(* IEC 61131-3 sources: B-R/Processes/EDT, 38 files *)

(* ---- EDTP1S1_1_ACTION.st ---- *)
ACTION P1S1_1_ACT:
	//步与步之间切换的设定时间,至少设置为5s(可更改，调整阀门到位、液位延时后),用于检查步骤错误信号
	FOR i := 0 TO EDTP1S1_1_STEP_NUM DO
		IF EDTP1S1_1_ST[i] < T#5s THEN
			EDTP1S1_1_ST[i] := T#5s;
		END_IF;
		EDTP1S1_1_STEP[i].set_time := EDTP1S1_1_ST[i];
	END_FOR;

	//流程步骤
	ProcessHandleFC(EDTP1S1_1,EDTP1S1_1_STEP[0],EDTP1S1_1_STEP_NUM);

	//object 手自动切换
	IF (EDTP1S1_1.status.mode <> 0) AND (NOT EDTP1S1_1.auto_mode_edge) THEN
		EDTP1S1_1.auto_mode_edge := TRUE;
		EDTP1S1_1.manual_mode_edge := FALSE;
		EDTR01.control.auto_operate := TRUE;
		EDTFQV0502.control.auto_operate := TRUE;
		EDTXV0505.control.auto_operate := TRUE;
	END_IF;

	IF (EDTP1S1_1.status.mode = 0) AND (NOT EDTP1S1_1.manual_mode_edge) THEN
		EDTP1S1_1.manual_mode_edge := TRUE;
		EDTP1S1_1.auto_mode_edge := FALSE;
		EDTR01.control.manual_operate := TRUE;
		EDTFQV0502.control.manual_operate := TRUE;
		EDTXV0505.control.manual_operate := TRUE;
	END_IF;

	//错误信号停机
	EDTP1S1_1.input.error_signal := (EDTR01.status.motor_status >= 2) OR (EDTFQV0502.status.valve_status >= 2) OR
	(EDTXV0505.status.valve_status >= 2);

	//步骤执行动作
	IF EDTP1S1_1.status.run_state = 1 THEN
		CASE EDTP1S1_1.status.run_step OF
			0:
				//初始化检查
				IF NOT EDTP1S1_1_STEP[0].done THEN
					EDTR01.control.auto_operate := TRUE;
					EDTFQV0502.control.auto_operate := TRUE;
					EDTXV0505.control.auto_operate := TRUE;
					EDTP1S1_1_STEP[0].done := TRUE;
				END_IF;
			1:
				//关闭底阀
				EDTXV0505.input.auto_open_signal := FALSE;
				IF EDTXV0505.input.close_feedback_state THEN
					EDTP1S1_1_STEP[1].done := TRUE;
				END_IF;
			2:
				//加定量纯水
				LiquidTransfer_3(sp_time := DINT_TO_TIME(EDTP1S1_1_PARA_T1 * 1000),
				sp_accumulation := EDTP1S1_1_PARA_AC1,
				done := EDTP1S1_1_STEP[2].done,
				flowmeter := EDTFQIT1904);
				EDTFQV0502.input.auto_open_signal := LiquidTransfer_3.run;
			3:
				//开启搅拌
				EDTR01.input.auto_run_signal := TRUE;
				IF EDTR01.input.run_feedback THEN
					EDTP1S1_1_STEP[3].done := TRUE;
				END_IF;
			4:
				//人工投料，完成后点击确认
			5:
				//溶解计时
				TON_41.PT := DINT_TO_TIME(EDTP1S1_1_PARA_T2 * 60 * 1000);
				TON_41.IN := TRUE;
				IF TON_41.Q THEN
					TON_41.IN := FALSE;
					EDTP1S1_1_STEP[5].done := TRUE;
				END_IF;
				TON_41();
			6:
				//观察溶解结束后点击确认
		END_CASE;
	END_IF;

	//人工确认步骤可用
	IF (EDTP1S1_1.status.run_state) AND (NOT EDTP1S1_1_STEP[EDTP1S1_1.status.run_step].done AND ((EDTP1S1_1.status.run_step = 4) OR (EDTP1S1_1.status.run_step = 6))) THEN
		EDTP1S1_1.status.confirm_enable := TRUE;
	ELSE
		EDTP1S1_1.status.confirm_enable := FALSE;
	END_IF;
END_ACTION

(* ---- EDTP1S1_ACTION.st ---- *)
ACTION P1S1_ACT:
	//步与步之间切换的设定时间,至少设置为5s(可更改，调整阀门到位、液位延时后),用于检查步骤错误信号
	FOR i := 0 TO EDTP1S1_STEP_NUM DO
		IF EDTP1S1_ST[i] < T#5s THEN
			EDTP1S1_ST[i] := T#5s;
		END_IF;
		EDTP1S1_STEP[i].set_time := EDTP1S1_ST[i];
	END_FOR;

	//流程步骤
	ProcessHandleFC(EDTP1S1,EDTP1S1_STEP[0],EDTP1S1_STEP_NUM);

	//object 手自动切换
	IF (EDTP1S1.status.mode <> 0) AND (NOT EDTP1S1.auto_mode_edge) THEN
		EDTP1S1.auto_mode_edge := TRUE;
		EDTP1S1.manual_mode_edge := FALSE;
		EDTR02.control.auto_operate := TRUE;
		EDTFQV0101.control.auto_operate := TRUE;
		EDTXV0102.control.auto_operate := TRUE;
	END_IF;

	IF (EDTP1S1.status.mode = 0) AND (NOT EDTP1S1.manual_mode_edge) THEN
		EDTP1S1.manual_mode_edge := TRUE;
		EDTP1S1.auto_mode_edge := FALSE;
		EDTR02.control.manual_operate := TRUE;
		EDTFQV0101.control.manual_operate := TRUE;
		EDTXV0102.control.manual_operate := TRUE;
	END_IF;

	//错误信号停机
	EDTP1S1.input.error_signal := (EDTR02.status.motor_status >= 2) OR (EDTFQV0101.status.valve_status >= 2) OR
	(EDTXV0102.status.valve_status >= 2);

	//步骤执行动作
	IF EDTP1S1.status.run_state = 1 THEN
		CASE EDTP1S1.status.run_step OF
			0:
				//初始化检查
				IF NOT EDTP1S1_STEP[0].done THEN
					EDTR02.control.auto_operate := TRUE;
					EDTFQV0101.control.auto_operate := TRUE;
					EDTXV0102.control.auto_operate := TRUE;
					EDTP1S1_STEP[0].done := TRUE;
				END_IF;
			1:
				//关底阀
				EDTXV0102.input.auto_open_signal := FALSE;
				IF EDTXV0102.input.close_feedback_state THEN
					EDTP1S1_STEP[1].done := TRUE;
				END_IF;
			2:
				//加定量纯水
				LiquidTransfer_0(sp_time := DINT_TO_TIME(EDTP1S1_PARA_T1 * 1000),
				sp_accumulation := EDTP1S1_PARA_AC1,
				done := EDTP1S1_STEP[2].done,
				flowmeter := EDTFQIT1904);
				EDTFQV0101.input.auto_open_signal := LiquidTransfer_0.run;
			3:
				//开启搅拌
				EDTR02.input.auto_run_signal := TRUE;
				IF EDTR02.input.run_feedback THEN
					EDTP1S1_STEP[3].done := TRUE;
				END_IF;
			4:
				//人工投料，完成后点击确认
			5:
				//溶解计时
				TON_49.PT := DINT_TO_TIME(EDTP1S1_PARA_T2 * 60 * 1000);
				TON_49.IN := TRUE;
				IF TON_49.Q THEN
					TON_49.IN := FALSE;
					EDTP1S1_STEP[5].done := TRUE;
				END_IF;
				TON_49();
			6:
				//观察溶解结束
			7:
				//开底阀，关搅拌
				EDTXV0102.input.auto_open_signal := TRUE;
				IF EDTXV0102.input.open_feedback_state THEN
					EDTR02.input.auto_run_signal := FALSE;
					IF NOT EDTR02.input.run_feedback THEN
						EDTP1S1_STEP[7].done := TRUE;
					END_IF;
				END_IF;
			8:
				//观察釜内放料完成，点击确认
			9:
				EDTXV0102.input.auto_open_signal := FALSE;
				IF EDTXV0102.input.close_feedback_state THEN
					EDTP1S1_STEP[9].done := TRUE;
				END_IF;
			10:
				//手动通氮气清理过滤器
		END_CASE;
	END_IF;

	//人工确认步骤可用
	IF (EDTP1S1.status.run_state) AND (NOT EDTP1S1_STEP[EDTP1S1.status.run_step].done AND ((EDTP1S1.status.run_step = 4) OR (EDTP1S1.status.run_step = 6)
		OR (EDTP1S1.status.run_step = 8) OR (EDTP1S1.status.run_step = 10))) THEN
		EDTP1S1.status.confirm_enable := TRUE;
	ELSE
		EDTP1S1.status.confirm_enable := FALSE;
	END_IF;
END_ACTION

(* ---- EDTP1S2A_ACTION.st ---- *)
ACTION P1S2A_ACT:
	//设定时间
	FOR i := 0 TO EDTP1S2_STEP_NUM DO
		IF EDTP1S2A_ST[i] < T#5s THEN
			EDTP1S2A_ST[i] := T#5s;
		END_IF;
		EDTP1S2A_STEP[i].set_time := EDTP1S2A_ST[i];
	END_FOR;

	//流程步骤
	ProcessHandleFC(EDTP1S2A,EDTP1S2A_STEP[0],EDTP1S2_STEP_NUM);

	//object 手自动切换
	IF (EDTP1S2A.status.mode <> 0) AND (NOT EDTP1S2A.auto_mode_edge) THEN

		EDTP1S2A.auto_mode_edge := TRUE;
		EDTP1S2A.manual_mode_edge := FALSE;

		EDTP01.control.auto_operate := TRUE;
		EDTXV0205.control.auto_operate := TRUE;
		STFLV0701.control.auto_operate := TRUE;
		STFLV0702.control.auto_operate := TRUE;
		EDTLV0201.control.auto_operate := TRUE;
		STFP07.control.auto_operate := TRUE;
		EDTR07A.control.auto_operate := TRUE;
		EDTTV0201A.control.auto_operate := TRUE;
		EDTTV0201B.control.auto_operate := TRUE;
		EDTXV0201.control.auto_operate := TRUE;
		EDTXV0204.control.auto_operate := TRUE;
		EDTXV0505.control.auto_operate := TRUE;
		EDTFQV0203A.control.auto_operate := TRUE;
		EDTP26.control.auto_operate := TRUE;
	END_IF;

	IF (EDTP1S2A.status.mode = 0) AND (NOT EDTP1S2A.manual_mode_edge) THEN

		EDTP1S2A.manual_mode_edge := TRUE;
		EDTP1S2A.auto_mode_edge := FALSE;

		EDTP01.control.manual_operate := TRUE;
		EDTXV0205.control.manual_operate := TRUE;
		STFLV0701.control.manual_operate := TRUE;
		STFLV0702.control.manual_operate := TRUE;
		EDTLV0201.control.manual_operate := TRUE;
		STFP07.control.manual_operate := TRUE;
		EDTR07A.control.manual_operate := TRUE;
		EDTTV0201A.control.manual_operate := TRUE;
		EDTTV0201B.control.manual_operate := TRUE;
		EDTXV0201.control.manual_operate := TRUE;
		EDTXV0204.control.manual_operate := TRUE;
		EDTXV0505.control.manual_operate := TRUE;
		EDTFQV0203A.control.manual_operate := TRUE;
		EDTP26.control.manual_operate := TRUE;
	END_IF;

	//错误信号停机
	EDTP1S2A.input.error_signal := (EDTP01.status.motor_status >= 2) OR (EDTXV0205.status.valve_status >= 2) OR
	(STFLV0701.status.valve_status >= 2) OR (STFLV0702.status.valve_status >= 2) OR (EDTLV0201.status.valve_status >= 2) OR
	(STFP07.status.motor_status >= 2) OR (EDTR07A.status.motor_status >= 2) OR
	(EDTTV0201A.status.valve_status >= 2) OR (EDTTV0201B.status.valve_status >= 2) OR (EDTXV0201.status.valve_status >= 2) OR
	(EDTP26.status.motor_status >= 2) OR (EDTFQV0203A.status.valve_status >= 2) OR (EDTXV0505.status.valve_status >= 2) OR
	(EDTXV0204.status.valve_status >= 2);

	IF EDTP1S2A.status.run_state = 1 THEN
		CASE EDTP1S2A.status.run_step OF
			0:
				//初始化
				IF NOT EDTP1S2A_STEP[0].done THEN
					EDTP01.control.auto_operate := TRUE;
					EDTXV0205.control.auto_operate := TRUE;
					STFLV0701.control.auto_operate := TRUE;
					STFLV0702.control.auto_operate := TRUE;
					EDTLV0201.control.auto_operate := TRUE;
					STFP07.control.auto_operate := TRUE;
					EDTR07A.control.auto_operate := TRUE;
					EDTTV0201A.control.auto_operate := TRUE;
					EDTTV0201B.control.auto_operate := TRUE;
					EDTXV0201.control.auto_operate := TRUE;
					EDTXV0204.control.auto_operate := TRUE;
					EDTXV0505.control.auto_operate := TRUE;
					EDTFQV0203A.control.auto_operate := TRUE;
					EDTP26.control.auto_operate := TRUE;
					EDTP1S2A_STEP[0].done := TRUE;
				END_IF;
			1:
				//人工确认投料
			2:
				//滴加
				CASE p1_step2_2a OF
					0:
						IF NOT EDTP1S2A_STEP[2].done THEN
							p1_step2_2a := 1;
						END_IF;
					1:
						EDTXV0201.input.auto_open_signal := TRUE;
						EDTR07A.input.auto_run_signal := TRUE;
						IF EDTXV0201.input.open_feedback_state AND EDTR07A.input.run_feedback THEN
							p1_step2_2a := 2;
						END_IF;
					2:
						IF EDTTIT0201.status.value <= EDTP1S2_PARA_Temp1 THEN
							p1_step2_2a := 3;
						END_IF;
					3:
						TON_2.PT := DINT_TO_TIME(EDTP1S2_PARA_T5 * 60 * 1000);
						TON_2.IN := TRUE;
						IF EDTTIT0201.status.value <= EDTP1S2_PARA_Temp2 THEN
							EDTTV0201A.input.auto_open_signal := TRUE;
							EDTTV0201B.input.auto_open_signal := TRUE;
						END_IF;
						IF EDTTIT0201.status.value >= EDTP1S2_PARA_Temp3 THEN
							EDTTV0201A.input.auto_open_signal := FALSE;
							EDTTV0201B.input.auto_open_signal := FALSE;
						END_IF;
						IF TON_2.Q THEN
							TON_2.IN := FALSE;
							EDTXV0201.input.auto_open_signal := FALSE;
							EDTTV0201A.input.auto_open_signal := TRUE;
							EDTTV0201B.input.auto_open_signal := TRUE;
							p1_step2_2a := 4;
						END_IF;
					4:
						TON_2.PT := DINT_TO_TIME(EDTP1S2_PARA_T6 * 60 * 1000);
						TON_2.IN := TRUE;
						IF TON_2.Q THEN
							TON_2.IN := FALSE;
							EDTTV0201A.input.auto_open_signal := FALSE;
							EDTTV0201B.input.auto_open_signal := FALSE;
							p1_step2_2a := 5;
						END_IF;
					5:
						IF EDTTV0201A.input.close_feedback_state AND EDTTV0201B.input.close_feedback_state THEN
							EDTP1S2A_STEP[2].done := TRUE;
							p1_step2_2a := 0;
						END_IF;
				END_CASE;
				TON_2();
			3:
				//取样确认
			4:
				TON_9.PT := DINT_TO_TIME(EDTP1S2_PARA_T7 * 60 * 1000);
				EDTR07A.input.auto_run_signal := FALSE;
				IF NOT EDTR07A.input.run_feedback THEN
					TON_9.IN := TRUE;
				END_IF;
				IF TON_9.Q THEN
					TON_9.IN := FALSE;
					EDTP1S2A_STEP[4].done := TRUE;
				END_IF;
				TON_9();
		END_CASE;
	END_IF;

	//R07A进ABC溶液
	IF r07a_add THEN
		CASE p1_step2_4a OF
			0:
				EDTXV0204.input.auto_open_signal := FALSE;
				EDTXV0201.input.auto_open_signal := TRUE;
				IF EDTXV0204.input.close_feedback_state AND EDTXV0201.input.open_feedback_state THEN
					p1_step2_4a := 1;
				END_IF;
			1:
				EDTXV0505.input.auto_open_signal := TRUE;
				EDTFQV0203A.input.auto_open_signal := TRUE;
				IF EDTXV0505.input.open_feedback_state AND EDTFQV0203A.input.open_feedback_state THEN
					p1_step2_4a := 2;
				END_IF;
			2:
			//等待液体充满泵后，再启动P26防止抽空。
				TON_54.PT := DINT_TO_TIME(EDTP1S2A_PARA_T4 * 1000);
				TON_54.IN := TRUE;
				IF TON_54.Q THEN
					TON_54.IN := FALSE;
					p1_step2_4a := 3;
				END_IF;
			3:
				LiquidTransfer_4(sp_time := DINT_TO_TIME(EDTP1S2A_PARA_T8 * 1000),
				sp_accumulation := EDTP1S2A_PARA_AC2,
				done := p1_step2_4a_3_done,
				flowmeter := EDTFQIT0203);
				EDTP26.input.auto_run_signal := LiquidTransfer_4.run;
				IF p1_step2_4a_3_done AND (NOT EDTP26.input.run_feedback) AND (NOT EDTP26.input.auto_run_signal) THEN
					p1_step2_4a := 4;
					p1_step2_4a_3_done := FALSE;
				END_IF;
			4:
				IF EDTFQIT0203.flowrate <= flowrate_threshold THEN
					EDTXV0505.input.auto_open_signal := FALSE;
					EDTFQV0203A.input.auto_open_signal := FALSE;
				END_IF;
				IF EDTXV0505.input.close_feedback_state AND EDTFQV0203A.input.close_feedback_state THEN
					r07a_add := FALSE;
					p1_step2_4a := 0;
				END_IF;
		END_CASE;
		TON_54();
	END_IF;

	//V02A（SSS溶液）进料
	IF v02a_add THEN
		CASE p1_step2_1a OF
			0:
				p1_step2_1a := 1;
			1:
				EDTXV0205.input.auto_open_signal := TRUE;
				IF EDTXV0205.input.open_feedback_state THEN
					p1_step2_1a := 2;
				END_IF;
			2:
				LiquidAddSimple_0(level_value := EDTLIT0203.status.value,
				sp_value := EDTP1S2A_PARA_L2,
				sp_time := DINT_TO_TIME(EDTP1S2A_PARA_T1 * 60 * 1000),
				done := p1_step2_1a_2_done);
				EDTP01.input.auto_run_signal := LiquidAddSimple_0.run;
				IF p1_step2_1a_2_done AND (NOT EDTP01.input.run_feedback) AND (NOT EDTP01.input.auto_run_signal) THEN
					p1_step2_1a := 3;
					p1_step2_1a_2_done := FALSE;
				END_IF;
			3:
				TON_1.PT := DINT_TO_TIME(EDTP1S2A_PARA_T2 * 1000);
				TON_1.IN := TRUE;
				IF TON_1.Q THEN
					TON_1.IN := FALSE;
					p1_step2_1a := 4;
				END_IF;
			4:
				EDTXV0205.input.auto_open_signal := FALSE;
				IF EDTXV0205.input.close_feedback_state THEN
					v02a_add := FALSE;
					p1_step2_1a := 0;
				END_IF;
		END_CASE;
		TON_1();
	END_IF;

	//V03A（MCE）进料
	IF v03a_add THEN
		CASE p1_step2_3a OF
			0:
				p1_step2_3a := 1;
			1:
				STFLV0702.input.auto_open_signal := FALSE;
				STFLV0701.input.auto_open_signal := FALSE;
				EDTLV0201.input.auto_open_signal := TRUE;
				IF EDTLV0201.input.open_feedback_state AND STFLV0701.input.close_feedback_state
					AND STFLV0702.input.close_feedback_state THEN
					p1_step2_3a := 2;
				END_IF;
			2:
				LiquidAdd_3(level_value := EDTLIT0201.status.value,
				sp_value := EDTP1S2A_PARA_L1,
				sp_accumulation := EDTP1S2A_PARA_AC1,
				sp_time := DINT_TO_TIME(EDTP1S2A_PARA_T3 * 1000),
				flowmeter := STFFQIT0702,
				done := p1_step2_3a_2_done);
				STFP07.input.auto_run_signal := LiquidAdd_3.run;
				IF p1_step2_3a_2_done AND (NOT STFP07.input.run_feedback) AND (NOT STFP07.input.auto_run_signal) THEN
					p1_step2_3a := 3;
				END_IF;
			3:
				IF STFFQIT0702.flowrate <= flowrate_threshold THEN
					EDTLV0201.input.auto_open_signal := FALSE;
				END_IF;
				IF EDTLV0201.input.close_feedback_state THEN
					p1_step2_3a_2_done := FALSE;
					p1_step2_3a := 0;
					v03a_add := FALSE;
				END_IF;
		END_CASE;
	END_IF;
		//人工确认步骤可用
		IF (EDTP1S2A.status.run_state) AND (NOT EDTP1S2A_STEP[EDTP1S2A.status.run_step].done AND ((EDTP1S2A.status.run_step = 1) OR (EDTP1S2A.status.run_step = 3))) THEN
			EDTP1S2A.status.confirm_enable := TRUE;
		ELSE
			EDTP1S2A.status.confirm_enable := FALSE;
		END_IF;
		END_ACTION

(* ---- EDTP1S2B_ACTION.st ---- *)
ACTION P1S2B_ACT:
	//设定时间
	FOR i := 0 TO EDTP1S2_STEP_NUM DO
		IF EDTP1S2B_ST[i] < T#5s THEN
			EDTP1S2B_ST[i] := T#5s;
		END_IF;
		EDTP1S2B_STEP[i].set_time := EDTP1S2B_ST[i];
	END_FOR;

	//流程步骤
	ProcessHandleFC(EDTP1S2B,EDTP1S2B_STEP[0],EDTP1S2_STEP_NUM);

	//object 手自动切换
	IF (EDTP1S2B.status.mode <> 0) AND (NOT EDTP1S2B.auto_mode_edge) THEN

		EDTP1S2B.auto_mode_edge := TRUE;
		EDTP1S2B.manual_mode_edge := FALSE;

		EDTP01.control.auto_operate := TRUE;
		EDTXV0206.control.auto_operate := TRUE;
		STFLV0701.control.auto_operate := TRUE;
		STFLV0702.control.auto_operate := TRUE;
		EDTLV0202.control.auto_operate := TRUE;
		STFP07.control.auto_operate := TRUE;
		EDTR07B.control.auto_operate := TRUE;
		EDTTV0202A.control.auto_operate := TRUE;
		EDTTV0202B.control.auto_operate := TRUE;
		EDTXV0202.control.auto_operate := TRUE;
		EDTXV0203.control.auto_operate := TRUE;
		EDTXV0505.control.auto_operate := TRUE;
		EDTFQV0203B.control.auto_operate := TRUE;
		EDTP26.control.auto_operate := TRUE;
	END_IF;

	IF (EDTP1S2B.status.mode = 0) AND (NOT EDTP1S2B.manual_mode_edge) THEN

		EDTP1S2B.manual_mode_edge := TRUE;
		EDTP1S2B.auto_mode_edge := FALSE;

		EDTP01.control.manual_operate := TRUE;
		EDTXV0206.control.manual_operate := TRUE;
		STFLV0701.control.manual_operate := TRUE;
		STFLV0702.control.manual_operate := TRUE;
		EDTLV0202.control.manual_operate := TRUE;
		STFP07.control.manual_operate := TRUE;
		EDTR07B.control.manual_operate := TRUE;
		EDTTV0202A.control.manual_operate := TRUE;
		EDTTV0202B.control.manual_operate := TRUE;
		EDTXV0202.control.manual_operate := TRUE;
		EDTXV0203.control.manual_operate := TRUE;
		EDTXV0505.control.manual_operate := TRUE;
		EDTFQV0203B.control.manual_operate := TRUE;
		EDTP26.control.manual_operate := TRUE;
	END_IF;

	//错误信号停机
	EDTP1S2B.input.error_signal := (EDTP01.status.motor_status >= 2) OR (EDTXV0206.status.valve_status >= 2) OR
	(STFLV0701.status.valve_status >= 2) OR (STFLV0702.status.valve_status >= 2) OR (EDTLV0202.status.valve_status >= 2) OR
	(STFP07.status.motor_status >= 2) OR (EDTR07B.status.motor_status >= 2) OR
	(EDTTV0202A.status.valve_status >= 2) OR (EDTTV0202B.status.valve_status >= 2) OR (EDTXV0202.status.valve_status >= 2) OR
	(EDTP26.status.motor_status >= 2) OR (EDTFQV0203B.status.valve_status >= 2) OR (EDTXV0505.status.valve_status >= 2) OR
	(EDTXV0203.status.valve_status >= 2);

	IF EDTP1S2B.status.run_state = 1 THEN
		CASE EDTP1S2B.status.run_step OF
			0:
				//初始化
				IF NOT EDTP1S2B_STEP[0].done THEN
					EDTP01.control.auto_operate := TRUE;
					EDTXV0206.control.auto_operate := TRUE;
					STFLV0701.control.auto_operate := TRUE;
					STFLV0702.control.auto_operate := TRUE;
					EDTLV0202.control.auto_operate := TRUE;
					STFP07.control.auto_operate := TRUE;
					EDTR07B.control.auto_operate := TRUE;
					EDTTV0202A.control.auto_operate := TRUE;
					EDTTV0202B.control.auto_operate := TRUE;
					EDTXV0202.control.auto_operate := TRUE;
					EDTXV0203.control.auto_operate := TRUE;
					EDTXV0505.control.auto_operate := TRUE;
					EDTFQV0203B.control.auto_operate := TRUE;
					EDTP26.control.auto_operate := TRUE;
					EDTP1S2B_STEP[0].done := TRUE;
				END_IF;
			1:
				//人工确认投料
			2:
				//滴加
				CASE p1_step2_2b OF
					0:
						IF NOT EDTP1S2B_STEP[2].done THEN
							p1_step2_2b := 1;
						END_IF;
					1:
						EDTXV0202.input.auto_open_signal := TRUE;
						EDTR07B.input.auto_run_signal := TRUE;
						IF EDTXV0202.input.open_feedback_state AND EDTR07B.input.run_feedback THEN
							p1_step2_2b := 2;
						END_IF;
					2:
						IF EDTTIT0202.status.value <= EDTP1S2_PARA_Temp1 THEN
							p1_step2_2b := 3;
						END_IF;
					3:
						TON_5.PT := DINT_TO_TIME(EDTP1S2_PARA_T5 * 60 * 1000);
						TON_5.IN := TRUE;
						IF EDTTIT0202.status.value <= EDTP1S2_PARA_Temp2 THEN
							EDTTV0202A.input.auto_open_signal := TRUE;
							EDTTV0202B.input.auto_open_signal := TRUE;
						END_IF;
						IF EDTTIT0202.status.value >= EDTP1S2_PARA_Temp3 THEN
							EDTTV0202A.input.auto_open_signal := FALSE;
							EDTTV0202B.input.auto_open_signal := FALSE;
						END_IF;
						IF TON_5.Q THEN
							TON_5.IN := FALSE;
							EDTXV0202.input.auto_open_signal := FALSE;
							EDTTV0202A.input.auto_open_signal := TRUE;
							EDTTV0202B.input.auto_open_signal := TRUE;
							p1_step2_2b := 4;
						END_IF;
					4:
						TON_5.PT := DINT_TO_TIME(EDTP1S2_PARA_T6 * 60 * 1000);
						TON_5.IN := TRUE;
						IF TON_5.Q THEN
							TON_5.IN := FALSE;
							EDTTV0202A.input.auto_open_signal := FALSE;
							EDTTV0202B.input.auto_open_signal := FALSE;
							p1_step2_2b := 5;
						END_IF;
					5:
						IF EDTTV0202A.input.close_feedback_state AND EDTTV0202B.input.close_feedback_state THEN
							EDTP1S2B_STEP[2].done := TRUE;
							p1_step2_2b := 0;
						END_IF;
				END_CASE;
				TON_5();
			3:
				//取样确认
			4:
				TON_18.PT := DINT_TO_TIME(EDTP1S2_PARA_T7 * 60 * 1000);
				EDTR07B.input.auto_run_signal := FALSE;
				IF NOT EDTR07B.input.run_feedback THEN
					TON_18.IN := TRUE;
				END_IF;
				IF TON_18.Q THEN
					TON_18.IN := FALSE;
					EDTP1S2B_STEP[4].done := TRUE;
				END_IF;
				TON_18();
		END_CASE;
	END_IF;

	//R07A进ABC溶液
	IF r07b_add THEN
		CASE p1_step2_4b OF
			0:
				EDTXV0203.input.auto_open_signal := FALSE;
				EDTXV0202.input.auto_open_signal := TRUE;
				IF EDTXV0203.input.close_feedback_state AND EDTXV0202.input.open_feedback_state THEN
					p1_step2_4b := 1;
				END_IF;
			1:
				EDTXV0505.input.auto_open_signal := TRUE;
				EDTFQV0203B.input.auto_open_signal := TRUE;
				IF EDTXV0505.input.open_feedback_state AND EDTFQV0203B.input.open_feedback_state THEN
					p1_step2_4b := 2;
				END_IF;
			2:
				//等待液体充满泵后，再启动P26防止抽空。
				TON_55.PT := DINT_TO_TIME(EDTP1S2B_PARA_T4 * 1000);
				TON_55.IN := TRUE;
				IF TON_55.Q THEN
					TON_55.IN := FALSE;
					p1_step2_4b := 3;
				END_IF;
			3:
				LiquidTransfer_5(sp_time := DINT_TO_TIME(EDTP1S2B_PARA_T8 * 1000),
				sp_accumulation := EDTP1S2B_PARA_AC2,
				done := p1_step2_4b_3_done,
				flowmeter := EDTFQIT0203);
				EDTP26.input.auto_run_signal := LiquidTransfer_5.run;
				IF p1_step2_4b_3_done AND (NOT EDTP26.input.run_feedback) AND (NOT EDTP26.input.auto_run_signal) THEN
					p1_step2_4b := 4;
					p1_step2_4b_3_done := FALSE;
				END_IF;
			4:
				IF EDTFQIT0203.flowrate <= flowrate_threshold THEN
					EDTXV0505.input.auto_open_signal := FALSE;
					EDTFQV0203B.input.auto_open_signal := FALSE;
				END_IF;
				IF EDTXV0505.input.close_feedback_state AND EDTFQV0203B.input.close_feedback_state THEN
					r07b_add := FALSE;
					p1_step2_4b := 0;
				END_IF;
		END_CASE;
		TON_55();
	END_IF;

	//V02B（SSS溶液）进料
	IF v02b_add THEN
		CASE p1_step2_1b OF
			0:
				p1_step2_1b := 1;
			1:
				EDTXV0206.input.auto_open_signal := TRUE;
				IF EDTXV0206.input.open_feedback_state THEN
					p1_step2_1b := 2;
				END_IF;
			2:
				LiquidAddSimple_1(level_value := EDTLIT0204.status.value,
				sp_value := EDTP1S2B_PARA_L2,
				sp_time := DINT_TO_TIME(EDTP1S2B_PARA_T1 * 60 * 1000),
				done := p1_step2_1b_2_done);
				EDTP01.input.auto_run_signal := LiquidAddSimple_1.run;
				IF p1_step2_1b_2_done AND (NOT EDTP01.input.run_feedback) AND (NOT EDTP01.input.auto_run_signal) THEN
					p1_step2_1b := 3;
					p1_step2_1b_2_done := FALSE;
				END_IF;
			3:
				TON_4.PT := DINT_TO_TIME(EDTP1S2B_PARA_T2 * 1000);
				TON_4.IN := TRUE;
				IF TON_4.Q THEN
					TON_4.IN := FALSE;
					p1_step2_1b := 4;
				END_IF;
			4:
				EDTXV0206.input.auto_open_signal := FALSE;
				IF EDTXV0206.input.close_feedback_state THEN
					v02b_add := FALSE;
					p1_step2_1b := 0;
				END_IF;
		END_CASE;
		TON_4();
	END_IF;

	//V03B（MCE）进料
	IF v03b_add THEN
		CASE p1_step2_3b OF
			0:
				p1_step2_3b := 1;
			1:
				STFLV0702.input.auto_open_signal := FALSE;
				STFLV0701.input.auto_open_signal := FALSE;
				EDTLV0202.input.auto_open_signal := TRUE;
				IF EDTLV0202.input.open_feedback_state AND STFLV0701.input.close_feedback_state
					AND STFLV0702.input.close_feedback_state THEN
					p1_step2_3b := 2;
				END_IF;
			2:
				LiquidAdd_5(level_value := EDTLIT0202.status.value,
				sp_value := EDTP1S2B_PARA_L1,
				sp_accumulation := EDTP1S2B_PARA_AC1,
				sp_time := DINT_TO_TIME(EDTP1S2B_PARA_T3 * 1000),
				flowmeter := STFFQIT0702,
				done := p1_step2_3b_2_done);
				STFP07.input.auto_run_signal := LiquidAdd_5.run;
				IF p1_step2_3b_2_done AND (NOT STFP07.input.run_feedback) AND (NOT STFP07.input.auto_run_signal) THEN
					p1_step2_3b := 3;
				END_IF;
			3:
				IF STFFQIT0702.flowrate <= flowrate_threshold THEN
					EDTLV0202.input.auto_open_signal := FALSE;
				END_IF;
				IF EDTLV0202.input.close_feedback_state THEN
					p1_step2_3b_2_done := FALSE;
					p1_step2_3b := 0;
					v03b_add := FALSE;
				END_IF;
		END_CASE;
	END_IF;

	//人工确认步骤可用
	IF (EDTP1S2B.status.run_state) AND (NOT EDTP1S2B_STEP[EDTP1S2B.status.run_step].done AND ((EDTP1S2B.status.run_step = 1) OR (EDTP1S2B.status.run_step = 3))) THEN
		EDTP1S2B.status.confirm_enable := TRUE;
	ELSE
		EDTP1S2B.status.confirm_enable := FALSE;
	END_IF;
		END_ACTION

(* ---- EDTP1S3_ACTION.st ---- *)
ACTION P1S3_ACT:
	//设定时间
	FOR i := 0 TO EDTP1S3_STEP_NUM DO
		IF EDTP1S3_ST[i] < T#5s THEN
			EDTP1S3_ST[i] := T#5s;
		END_IF;
		EDTP1S3_STEP[i].set_time := EDTP1S3_ST[i];
	END_FOR;

	//流程步骤
	ProcessHandleFC(EDTP1S3,EDTP1S3_STEP[0],EDTP1S3_STEP_NUM);

	//object 手自动切换
	IF (EDTP1S3.status.mode <> 0) AND (NOT EDTP1S3.auto_mode_edge) THEN
		EDTP1S3.auto_mode_edge := TRUE;
		EDTP1S3.manual_mode_edge := FALSE;

		EDTXV0304.control.auto_operate := TRUE;
		EDTXV0410.control.auto_operate := TRUE;
		EDTXV0302.control.auto_operate := TRUE;
		EDTTV0301G.control.auto_operate := TRUE;
		EDTR13.control.auto_operate := TRUE;
		EDTP03.control.auto_operate := TRUE;
		EDTTV0301C.control.auto_operate := TRUE;
		EDTTV0301D.control.auto_operate := TRUE;
		EDTTV0301E.control.auto_operate := TRUE;
		EDTTV0301F.control.auto_operate := TRUE;
		EDTTV0301A.control.auto_operate := TRUE;
		EDTTV0301B.control.auto_operate := TRUE;
		EDTPV0301.control.auto_operate := TRUE;
	END_IF;

	IF (EDTP1S3.status.mode = 0) AND (NOT EDTP1S3.manual_mode_edge) THEN
		EDTP1S3.manual_mode_edge := TRUE;
		EDTP1S3.auto_mode_edge := FALSE;

		EDTXV0304.control.manual_operate := TRUE;
		EDTXV0410.control.manual_operate := TRUE;
		EDTXV0302.control.manual_operate := TRUE;
		EDTTV0301G.control.manual_operate := TRUE;
		EDTR13.control.manual_operate := TRUE;
		EDTP03.control.manual_operate := TRUE;
		EDTTV0301C.control.manual_operate := TRUE;
		EDTTV0301D.control.manual_operate := TRUE;
		EDTTV0301E.control.manual_operate := TRUE;
		EDTTV0301F.control.manual_operate := TRUE;
		EDTTV0301A.control.manual_operate := TRUE;
		EDTTV0301B.control.manual_operate := TRUE;
		EDTPV0301.control.manual_operate := TRUE;
	END_IF;

	//错误信号停机
	EDTP1S3.input.error_signal :=
	(EDTXV0304.status.valve_status >= 2) OR (EDTXV0410.status.valve_status >= 2) OR (EDTXV0302.status.valve_status >= 2) OR
	(EDTTV0301G.status.valve_status >= 2) OR (EDTR13.status.motor_status >= 2) OR
	(EDTP03.status.motor_status >= 2) OR (EDTTV0301C.status.valve_status >= 2) OR
	(EDTTV0301D.status.valve_status >= 2) OR (EDTTV0301E.status.valve_status >= 2) OR
	(EDTTV0301F.status.valve_status >= 2) OR (EDTTV0301A.status.valve_status >= 2) OR
	(EDTTV0301B.status.valve_status >= 2) OR (EDTPV0301.status.valve_status >= 2);

	IF EDTP1S3.status.run_state = 1 THEN
		CASE EDTP1S3.status.run_step OF
			0:
				//初始化
				IF NOT EDTP1S3_STEP[0].done THEN
					EDTXV0302.control.auto_operate := TRUE;
					EDTXV0304.control.auto_operate := TRUE;
					EDTXV0410.control.auto_operate := TRUE;
					EDTTV0301G.control.auto_operate := TRUE;
					EDTR13.control.auto_operate := TRUE;
					EDTP03.control.auto_operate := TRUE;
					EDTTV0301C.control.auto_operate := TRUE;
					EDTTV0301D.control.auto_operate := TRUE;
					EDTTV0301E.control.auto_operate := TRUE;
					EDTTV0301F.control.auto_operate := TRUE;
					EDTTV0301A.control.auto_operate := TRUE;
					EDTTV0301B.control.auto_operate := TRUE;
					EDTPV0301.control.auto_operate := TRUE;
					EDTP1S3_STEP[0].done := TRUE;
				END_IF;
			1:
				//确认R13釜空闲,手动开阀进料
			2:
				EDTXV0302.input.auto_open_signal := TRUE;
				IF EDTXV0302.input.open_feedback_state THEN
					EDTXV0304.input.auto_open_signal := TRUE;
				END_IF;
				IF EDTXV0304.input.open_feedback_state THEN
					EDTTV0301G.input.auto_open_signal := TRUE;
				END_IF;
				IF EDTTV0301G.input.open_feedback_state THEN
					EDTXV0410.input.auto_open_signal := TRUE;
				END_IF;
				IF EDTXV0302.input.open_feedback_state AND EDTXV0304.input.open_feedback_state AND EDTTV0301G.input.open_feedback_state
					AND EDTXV0410.input.open_feedback_state THEN
					EDTR13.input.auto_run_signal := TRUE;
					EDTP03.input.auto_run_signal := TRUE;
					IF EDTR13.input.run_feedback AND EDTP03.input.run_feedback THEN
						EDTP1S3_STEP[2].done := TRUE;
					END_IF;
				END_IF;
			3:
				CASE p1_step3_3 OF
					0:
						IF NOT EDTP1S3_STEP[3].done THEN
							p1_step3_3 := 1;
						END_IF;
					1:
						HeatPot_0(ST1 := DINT_TO_TIME(EDTP1S3_PARA_T1 * 1000),
						ST2 := DINT_TO_TIME(EDTP1S3_PARA_T2 * 1000),
						V3 := EDTTV0301C,
						V4 := EDTTV0301D,
						V5 := EDTTV0301E,
						V6 := EDTTV0301F,
						done := p1_step3_3_1_done);
						IF p1_step3_3_1_done THEN
							p1_step3_3 := 2;
						END_IF;
					2:
						IF EDTTIT0301.status.value >= EDTP1S3_PARA_Temp1 THEN
							EDTTV0301C.input.auto_open_signal := FALSE;
							IF EDTTIT0301.status.value >= EDTP1S3_PARA_Temp2 THEN
								p1_step3_3 := 3;
							END_IF;
						END_IF;
					3:
						TON_40.PT := DINT_TO_TIME(EDTP1S3_PARA_T3 * 60 * 1000);
						TON_40.IN := TRUE;
						IF TON_40.Q THEN
							TON_40.IN := FALSE;
							EDTTV0301D.input.auto_open_signal := FALSE;
							EDTTV0301E.input.auto_open_signal := FALSE;
							p1_step3_3 := 4;
						END_IF;
					4:
						TON_40.PT := DINT_TO_TIME(EDTP1S3_PARA_T4 * 60 * 1000);
						TON_40.IN := TRUE;
						IF TON_40.Q THEN
							TON_40.IN := FALSE;
							EDTTV0301F.input.auto_open_signal := TRUE;
							p1_step3_3 := 5;
						END_IF;
					5:
						TON_40.PT := DINT_TO_TIME(EDTP1S3_PARA_T5 * 1000);
						TON_40.IN := TRUE;
						IF TON_40.Q THEN
							TON_40.IN := FALSE;
							EDTTV0301F.input.auto_open_signal := FALSE;
							p1_step3_3 := 6;
						END_IF;
					6:
						IF EDTTV0301C.input.close_feedback_state AND EDTTV0301D.input.close_feedback_state AND EDTTV0301E.input.close_feedback_state AND EDTTV0301F.input.close_feedback_state THEN
							p1_step3_3 := 0;
							p1_step3_3_1_done := FALSE;
							EDTP1S3_STEP[3].done := TRUE;
						END_IF;
				END_CASE;
				TON_40();
			4:
				CASE p1_step3_4 OF
					0:
						IF NOT EDTP1S3_STEP[4].done THEN
							p1_step3_4 := 1;
						END_IF;
					1:
						EDTTV0301A.input.auto_open_signal := TRUE;
						IF EDTTV0301A.input.open_feedback_state THEN
							EDTTV0301B.input.auto_open_signal := TRUE;
							IF EDTTV0301B.input.open_feedback_state THEN
								p1_step3_4 := 2;
							END_IF;
						END_IF;
					2:
						IF EDTTIT0301.status.value <= EDTP1S3_PARA_Temp4 THEN
							EDTPV0301.input.auto_open_signal := TRUE;
							p1_step3_4 := 3;
						END_IF;
					3:
						IF EDTPIT0301.status.value >= EDTP1S3_PARA_P1 THEN
							EDTTV0301G.input.auto_open_signal := FALSE;
							IF EDTTV0301G.input.close_feedback_state THEN
								EDTP03.input.auto_run_signal := FALSE;
								p1_step3_4 := 4;
							END_IF;
						END_IF;
					4:
						IF NOT EDTP03.input.run_feedback THEN
							EDTXV0410.input.auto_open_signal := FALSE;
							EDTXV0304.input.auto_open_signal := FALSE;
							EDTTV0301A.input.auto_open_signal := FALSE;
							EDTTV0301B.input.auto_open_signal := FALSE;
							p1_step3_4 := 5;
						END_IF;
					5:
						IF EDTPIT0301.status.value >= EDTP1S3_PARA_P2 THEN
							EDTXV0302.input.auto_open_signal := FALSE;
							EDTPV0301.input.auto_open_signal := FALSE;
							EDTR13.input.auto_run_signal := FALSE;
							EDTP1S3_STEP[4].done := TRUE;
							p1_step3_4 := 0;
						END_IF;
				END_CASE;
		END_CASE;
	END_IF;

	//人工确认步骤可用
	IF (EDTP1S3.status.run_state) AND (NOT EDTP1S3_STEP[EDTP1S3.status.run_step].done AND ((EDTP1S3.status.run_step = 1))) THEN
		EDTP1S3.status.confirm_enable := TRUE;
	ELSE
		EDTP1S3.status.confirm_enable := FALSE;
	END_IF;
END_ACTION

(* ---- EDTP1S4_ACTION.st ---- *)
ACTION P1S4_ACT:
	//设定时间
	FOR i := 0 TO EDTP1S4_STEP_NUM DO
		IF EDTP1S4_ST[i] < T#5s THEN
			EDTP1S4_ST[i] := T#5s;
		END_IF;
		EDTP1S4_STEP[i].set_time := EDTP1S4_ST[i];
	END_FOR;

	//流程步骤
	ProcessHandleFC(EDTP1S4,EDTP1S4_STEP[0],EDTP1S4_STEP_NUM);

	//object 手自动切换
	IF (EDTP1S4.status.mode <> 0) AND (NOT EDTP1S4.auto_mode_edge) THEN
		EDTP1S4.auto_mode_edge := TRUE;
		EDTP1S4.manual_mode_edge := FALSE;

		EDTLV0401.control.auto_operate := TRUE;
		STFP14.control.auto_operate := TRUE;
		STFLV1401.control.auto_operate := TRUE;
		STFLV1402.control.auto_operate := TRUE;
		EDTXV0404.control.auto_operate := TRUE;
		EDTXV0405.control.auto_operate := TRUE;
	END_IF;

	IF (EDTP1S4.status.mode = 0) AND (NOT EDTP1S4.manual_mode_edge) THEN
		EDTP1S4.manual_mode_edge := TRUE;
		EDTP1S4.auto_mode_edge := FALSE;

		EDTLV0401.control.manual_operate := TRUE;
		STFP14.control.manual_operate := TRUE;
		STFLV1401.control.manual_operate := TRUE;
		STFLV1402.control.manual_operate := TRUE;
		EDTXV0404.control.manual_operate := TRUE;
		EDTXV0405.control.manual_operate := TRUE;
	END_IF;

	//错误信号停机
	EDTP1S4.input.error_signal := (EDTXV0405.status.valve_status >= 2) OR (EDTXV0404.status.valve_status >= 2) OR (EDTLV0401.status.valve_status >= 2) OR
	(STFLV1401.status.valve_status >= 2) OR (STFLV1402.status.valve_status >= 2) OR (STFP14.status.motor_status >= 2);

	IF EDTP1S4.status.run_state = 1 THEN
		CASE EDTP1S4.status.run_step OF
			0:
				//初始化
				IF NOT EDTP1S4_STEP[0].done THEN
					EDTLV0401.control.auto_operate := TRUE;
					STFP14.control.auto_operate := TRUE;
					STFLV1401.control.auto_operate := TRUE;
					STFLV1402.control.auto_operate := TRUE;
					EDTXV0404.control.auto_operate := TRUE;
					EDTXV0405.control.auto_operate := TRUE;
					EDTP1S4_STEP[0].done := TRUE;
				END_IF;
		END_CASE;
	END_IF;

	//人工确认步骤可用
//	IF (EDTP1S4.status.run_step = 1) OR (EDTP1S4.status.run_step = 5) THEN
//		EDTP1S4.status.confirm_enable := TRUE;
//	ELSE
//		EDTP1S4.status.confirm_enable := FALSE;
//	END_IF;

	//v07放料
	IF v07_release_start THEN
		CASE v07_release_step OF
			0:
				EDTXV0404.control.auto_operate := TRUE;
				EDTXV0405.control.auto_operate := TRUE;

				EDTXV0405.input.auto_open_signal := TRUE;
				IF EDTXV0405.input.open_feedback_state THEN
					EDTXV0404.input.auto_open_signal := TRUE;
					IF EDTXV0404.input.open_feedback_state THEN
						v07_release_step := 1;
					END_IF;
				END_IF;
			1:
				TON_6.PT := DINT_TO_TIME(EDTP1S4_PARA_T1 * 60 * 1000);
				TON_6.IN := TRUE;
				IF TON_6.Q AND (EDTLIT0401.status.value <= 0.0) THEN
					TON_6.IN := FALSE;
					v07_release_step := 2;
				END_IF;
			2:
				EDTXV0404.input.auto_open_signal := FALSE;
				EDTXV0405.input.auto_open_signal := FALSE;
				IF EDTXV0404.input.close_feedback_state AND EDTXV0405.input.close_feedback_state THEN
					v07_release_step := 3;
				END_IF;
			3:
				v07_release_step := 0;
				v07_release_start := FALSE;
		END_CASE;
		TON_6();
	END_IF;

	//v07进料
	IF v07_add_start THEN
		CASE v07_add_step OF
			0:
				EDTLV0401.control.auto_operate := TRUE;
				STFP14.control.auto_operate := TRUE;
				STFLV1401.control.auto_operate := TRUE;
				STFLV1402.control.auto_operate := TRUE;
				EDTXV0404.control.auto_operate := TRUE;
				EDTXV0405.control.auto_operate := TRUE;

				EDTLV0401.input.auto_open_signal := TRUE;
				EDTXV0405.input.auto_open_signal := TRUE;
				STFLV1401.input.auto_open_signal := TRUE;
				STFLV1402.input.auto_open_signal := FALSE;
				IF EDTLV0401.input.open_feedback_state AND EDTXV0405.input.open_feedback_state AND
					STFLV1401.input.open_feedback_state AND STFLV1402.input.close_feedback_state THEN
					v07_add_step := 1;
				END_IF;
			1:
				LiquidAdd_4(level_value := EDTLIT0401.status.value,
				sp_value := EDTP1S4_PARA_L1,
				sp_accumulation := EDTP1S4_PARA_AC1,
				sp_time := DINT_TO_TIME(EDTP1S4_PARA_T2 * 1000),
				flowmeter := STFFQIT1402,
				done := v07_add_done);
				STFP14.input.auto_run_signal := LiquidAdd_4.run;
				IF v07_add_done AND (NOT STFP14.input.run_feedback) AND (NOT STFP14.input.auto_run_signal) THEN
					v07_add_step := 2;
				END_IF;
			2:
				IF STFFQIT1402.flowrate <= flowrate_threshold THEN
					EDTLV0401.input.auto_open_signal := FALSE;
					EDTXV0405.input.auto_open_signal := FALSE;
					v07_add_step := 3;
				END_IF;
			3:
				v07_add_step := 0;
				v07_add_done := FALSE;
				v07_add_start := FALSE;
		END_CASE;
	END_IF;
END_ACTION

(* ---- EDTP1S5_ACTION.st ---- *)
ACTION P1S5_ACT:
	//设定时间
	FOR i := 0 TO EDTP1S5_STEP_NUM DO
		IF EDTP1S5_ST[i] < T#5s THEN
			EDTP1S5_ST[i] := T#5s;
		END_IF;
		EDTP1S5_STEP[i].set_time := EDTP1S5_ST[i];
	END_FOR;

	//流程步骤
	ProcessHandleFC(EDTP1S5,EDTP1S5_STEP[0],EDTP1S5_STEP_NUM);

	//object 手自动切换
	IF (EDTP1S5.status.mode <> 0) AND (NOT EDTP1S5.auto_mode_edge) THEN
		EDTP1S5.auto_mode_edge := TRUE;
		EDTP1S5.manual_mode_edge := FALSE;

		EDTXV0406.control.auto_operate := TRUE;
		EDTXV0407.control.auto_operate := TRUE;
		EDTXV0410.control.auto_operate := TRUE;
		EDTTV0403G.control.auto_operate := TRUE;
		EDTR19.control.auto_operate := TRUE;
		EDTP03.control.auto_operate := TRUE;
		EDTTV0403A.control.auto_operate := TRUE;
		EDTTV0403B.control.auto_operate := TRUE;
		EDTTV0403C.control.auto_operate := TRUE;
		EDTTV0403D.control.auto_operate := TRUE;
		EDTTV0403E.control.auto_operate := TRUE;
		EDTTV0403F.control.auto_operate := TRUE;
		EDTXV0411.control.auto_operate := TRUE;
		EDTPV0401.control.auto_operate := TRUE;
	END_IF;

	IF (EDTP1S5.status.mode = 0) AND (NOT EDTP1S5.manual_mode_edge) THEN
		EDTP1S5.manual_mode_edge := TRUE;
		EDTP1S5.auto_mode_edge := FALSE;

		EDTXV0406.control.manual_operate := TRUE;
		EDTXV0407.control.manual_operate := TRUE;
		EDTXV0410.control.manual_operate := TRUE;
		EDTTV0403G.control.manual_operate := TRUE;
		EDTR19.control.manual_operate := TRUE;
		EDTP03.control.manual_operate := TRUE;
		EDTTV0403A.control.manual_operate := TRUE;
		EDTTV0403B.control.manual_operate := TRUE;
		EDTTV0403C.control.manual_operate := TRUE;
		EDTTV0403D.control.manual_operate := TRUE;
		EDTTV0403E.control.manual_operate := TRUE;
		EDTTV0403F.control.manual_operate := TRUE;
		EDTXV0411.control.manual_operate := TRUE;
		EDTPV0401.control.manual_operate := TRUE;
	END_IF;

	//错误信号停机
	EDTP1S5.input.error_signal := (EDTXV0406.status.valve_status >= 2) OR (EDTXV0407.status.valve_status >= 2) OR
	(EDTXV0410.status.valve_status >= 2) OR (EDTTV0403G.status.valve_status >= 2) OR
	(EDTR19.status.motor_status >= 2) OR (EDTP03.status.motor_status >= 2) OR (EDTTV0403A.status.valve_status >= 2) OR
	(EDTTV0403B.status.valve_status >= 2) OR (EDTTV0403C.status.valve_status >= 2) OR (EDTTV0403D.status.valve_status >= 2) OR
	(EDTTV0403E.status.valve_status >= 2) OR (EDTTV0403F.status.valve_status >= 2) OR (EDTXV0411.status.valve_status >= 2) OR
	(EDTPV0401.status.valve_status >= 2);

	IF EDTP1S5.status.run_state = 1 THEN
		//步骤执行动作
		CASE EDTP1S5.status.run_step OF
			0:
				//初始化
				IF NOT EDTP1S5_STEP[0].done THEN
					EDTXV0406.control.auto_operate := TRUE;
					EDTXV0407.control.auto_operate := TRUE;
					EDTXV0410.control.auto_operate := TRUE;
					EDTTV0403G.control.auto_operate := TRUE;
					EDTR19.control.auto_operate := TRUE;
					EDTP03.control.auto_operate := TRUE;
					EDTTV0403A.control.auto_operate := TRUE;
					EDTTV0403B.control.auto_operate := TRUE;
					EDTTV0403C.control.auto_operate := TRUE;
					EDTTV0403D.control.auto_operate := TRUE;
					EDTTV0403E.control.auto_operate := TRUE;
					EDTTV0403F.control.auto_operate := TRUE;
					EDTXV0411.control.auto_operate := TRUE;
					EDTPV0401.control.auto_operate := TRUE;
					EDTP1S5_STEP[0].done := TRUE;
				END_IF;
			1:
				//确认V07空闲
			2:
				EDTXV0405.input.auto_open_signal := FALSE;
				IF EDTXV0405.input.close_feedback_state THEN
					EDTXV0406.input.auto_open_signal := TRUE;
				END_IF;
				IF EDTXV0406.input.open_feedback_state THEN
					EDTXV0407.input.auto_open_signal := TRUE;
				END_IF;
				IF EDTXV0407.input.open_feedback_state THEN
					EDTXV0410.input.auto_open_signal := TRUE;
				END_IF;
				IF EDTXV0410.input.open_feedback_state THEN
					EDTTV0403G.input.auto_open_signal := TRUE;
				END_IF;
				IF EDTTV0403G.input.open_feedback_state THEN
					EDTXV0411.input.auto_open_signal := TRUE;
				END_IF;
				IF EDTXV0406.input.open_feedback_state AND EDTXV0407.input.open_feedback_state AND EDTXV0405.input.close_feedback_state
					AND EDTXV0410.input.open_feedback_state AND EDTTV0403G.input.open_feedback_state AND EDTXV0411.input.open_feedback_state THEN
					EDTR19.input.auto_run_signal := TRUE;
					EDTP03.input.auto_run_signal := TRUE;
					IF EDTR19.input.run_feedback AND EDTP03.input.run_feedback THEN
						EDTP1S5_STEP[2].done := TRUE;
					END_IF;
				END_IF;
			3:
				CASE p1_step5_3 OF
					0:
						IF NOT EDTP1S5_STEP[3].done THEN
							p1_step5_3 := 1;
						END_IF;
					1:
						HeatPot_13(ST1 := DINT_TO_TIME(EDTP1S5_PARA_T1 * 1000),
						ST2 := DINT_TO_TIME(EDTP1S5_PARA_T2 * 1000),
						V3 := EDTTV0403C,
						V4 := EDTTV0403D,
						V5 := EDTTV0403E,
						V6 := EDTTV0403F,
						done := p1_step5_3_1_done);
						IF p1_step5_3_1_done THEN
							p1_step5_3_1_done := FALSE;
							p1_step5_3 := 2;
						END_IF;
					2:
						IF EDTTIT0403.status.value >= EDTP1S5_PARA_Temp1 THEN
							EDTTV0403C.input.auto_open_signal := FALSE;
							IF EDTTIT0403.status.value >= EDTP1S5_PARA_Temp2 THEN
								p1_step5_3 := 3;
							END_IF;
						END_IF;
					3:
						TON_45.PT := DINT_TO_TIME(EDTP1S5_PARA_T3 * 60 * 1000);
						TON_45.IN := TRUE;
						IF TON_45.Q THEN
							TON_45.IN := FALSE;
							EDTTV0403D.input.auto_open_signal := FALSE;
							EDTTV0403E.input.auto_open_signal := FALSE;
							p1_step5_3 := 4;
						END_IF;
					4:
						TON_45.PT := DINT_TO_TIME(EDTP1S5_PARA_T4 * 60 * 1000);
						TON_45.IN := TRUE;
						IF TON_45.Q THEN
							TON_45.IN := FALSE;
							EDTTV0403F.input.auto_open_signal := TRUE;
							p1_step5_3 := 5;
						END_IF;
					5:
						TON_45.PT := DINT_TO_TIME(EDTP1S5_PARA_T5 * 1000);
						TON_45.IN := TRUE;
						IF TON_45.Q THEN
							TON_45.IN := FALSE;
							EDTTV0403F.input.auto_open_signal := FALSE;
							p1_step5_3 := 6;
						END_IF;
					6:
						IF EDTTV0403C.input.close_feedback_state AND EDTTV0403D.input.close_feedback_state AND EDTTV0403E.input.close_feedback_state AND EDTTV0403F.input.close_feedback_state THEN
							EDTP1S5_STEP[3].done := TRUE;
							p1_step5_3 := 0;
						END_IF;
				END_CASE;
				TON_45();
			4:
				CASE p1_step5_4 OF
					0:
						IF NOT EDTP1S5_STEP[4].done THEN
							p1_step5_4 := 1;
						END_IF;
					1:
						EDTTV0403A.input.auto_open_signal := TRUE;
						IF	EDTTV0403A.input.open_feedback_state THEN
							EDTTV0403B.input.auto_open_signal := TRUE;
							IF EDTTV0403B.input.open_feedback_state THEN
								p1_step5_4 := 2;
							END_IF;
						END_IF;
					2:
						IF EDTTIT0403.status.value <= EDTP1S5_PARA_Temp4 THEN
							EDTPV0401.input.auto_open_signal := TRUE;
							p1_step5_4 := 3;
						END_IF;
					3:
						IF EDTPIT0401.status.value >= EDTP1S5_PARA_P1 THEN
							EDTTV0403G.input.auto_open_signal := FALSE;
							EDTP03.input.auto_run_signal := FALSE;
							EDTXV0406.input.auto_open_signal := FALSE;
							EDTXV0407.input.auto_open_signal := FALSE;
							EDTXV0410.input.auto_open_signal := FALSE;
							EDTTV0403A.input.auto_open_signal := FALSE;
							EDTTV0403B.input.auto_open_signal := FALSE;
							p1_step5_4 := 4;
						END_IF;
					4:
						IF EDTPIT0401.status.value >= EDTP1S5_PARA_P2 THEN
							EDTPV0401.input.auto_open_signal := FALSE;
							EDTXV0411.input.auto_open_signal := FALSE;
							EDTR19.input.auto_run_signal := FALSE;
							p1_step5_4 := 5;
						END_IF;
					5:
						EDTP1S5_STEP[4].done := TRUE;
						p1_step5_4 := 0;
				END_CASE;
		END_CASE;
	END_IF;

	//人工确认步骤可用
	IF (EDTP1S5.status.run_state) AND (NOT EDTP1S5_STEP[EDTP1S5.status.run_step].done AND ((EDTP1S5.status.run_step = 1))) THEN
		EDTP1S5.status.confirm_enable := TRUE;
	ELSE
		EDTP1S5.status.confirm_enable := FALSE;
	END_IF;
END_ACTION

(* ---- EDTP2S1_ACTION.st ---- *)
ACTION P2S1_ACT:
	//设定时间
	FOR i := 0 TO EDTP2S1_STEP_NUM DO
		IF EDTP2S1_ST[i] < T#5s THEN
			EDTP2S1_ST[i] := T#5s;
		END_IF;
		EDTP2S1_STEP[i].set_time := EDTP2S1_ST[i];
	END_FOR;

	//流程步骤
	ProcessHandleFC(EDTP2S1,EDTP2S1_STEP[0],EDTP2S1_STEP_NUM);

	//object 手自动切换
	IF (EDTP2S1.status.mode <> 0) AND (NOT EDTP2S1.auto_mode_edge) THEN
		EDTP2S1.auto_mode_edge := TRUE;
		EDTP2S1.manual_mode_edge := FALSE;

		EDTPV0501.control.auto_operate := TRUE;
		EDTXV0508.control.auto_operate := TRUE;
		EDTXV0501.control.auto_operate := TRUE;
		EDTXV0504.control.auto_operate := TRUE;
		EDTR01.control.auto_operate := TRUE;
		EDTFQV0501.control.auto_operate := TRUE;
		EDTP06.control.auto_operate := TRUE;
		EDTP05.control.auto_operate := TRUE;
		EDTXV0503.control.auto_operate := TRUE;
		EDTXV0507.control.auto_operate := TRUE;
		EDTXV0505.control.auto_operate := TRUE;
	END_IF;

	IF (EDTP2S1.status.mode = 0) AND (NOT EDTP2S1.manual_mode_edge) THEN
		EDTP2S1.manual_mode_edge := TRUE;
		EDTP2S1.auto_mode_edge := FALSE;

		EDTPV0501.control.manual_operate := TRUE;
		EDTXV0508.control.manual_operate := TRUE;
		EDTXV0501.control.manual_operate := TRUE;
		EDTXV0504.control.manual_operate := TRUE;
		EDTR01.control.manual_operate := TRUE;
		EDTFQV0501.control.manual_operate := TRUE;
		EDTP06.control.manual_operate := TRUE;
		EDTP05.control.manual_operate := TRUE;
		EDTXV0503.control.manual_operate := TRUE;
		EDTXV0507.control.manual_operate := TRUE;
		EDTXV0505.control.manual_operate := TRUE;
	END_IF;

	//错误信号停机
	EDTP2S1.input.error_signal := (EDTPV0501.status.valve_status >= 2) OR (EDTXV0508.status.valve_status >= 2) OR
	(EDTXV0501.status.valve_status >= 2) OR (EDTXV0504.status.valve_status >= 2) OR (EDTR01.status.motor_status >= 2) OR
	(EDTFQV0501.status.valve_status >= 2) OR (EDTP06.status.motor_status >= 2) OR (EDTP05.status.motor_status >= 2) OR
	(EDTXV0503.status.valve_status >= 2) OR (EDTXV0507.status.valve_status >= 2) OR (EDTXV0505.status.valve_status >= 2);

	IF EDTP2S1.status.run_state = 1 THEN
		CASE EDTP2S1.status.run_step OF
			0:
				//初始化
				IF NOT EDTP2S1_STEP[0].done THEN
					EDTPV0501.control.auto_operate := TRUE;
					EDTXV0508.control.auto_operate := TRUE;
					EDTXV0501.control.auto_operate := TRUE;
					EDTXV0504.control.auto_operate := TRUE;
					EDTR01.control.auto_operate := TRUE;
					EDTFQV0501.control.auto_operate := TRUE;
					EDTP06.control.auto_operate := TRUE;
					EDTP05.control.auto_operate := TRUE;
					EDTXV0503.control.auto_operate := TRUE;
					EDTXV0507.control.auto_operate := TRUE;
					EDTXV0505.control.auto_operate := TRUE;
					EDTP2S1_STEP[0].done := TRUE;
				END_IF;
			1:
				//确认V17液位
			2:
				CASE p2_step1_2 OF
					0:
						IF NOT EDTP2S1_STEP[2].done THEN
							p2_step1_2 := 1;
						END_IF;
					1:
						EDTXV0508.input.auto_open_signal := TRUE;
						EDTXV0504.input.auto_open_signal := TRUE;
						EDTXV0501.input.auto_open_signal := TRUE;
						IF EDTXV0508.input.open_feedback_state AND EDTXV0504.input.open_feedback_state AND EDTXV0501.input.open_feedback_state THEN
							p2_step1_2 := 2;
						END_IF;
					2:
						EDTFQV0501.input.auto_open_signal := TRUE;
						IF EDTFQV0501.input.open_feedback_state THEN
							p2_step1_2 := 3;
						END_IF;
					3:
						LiquidReleaseAdvanced_0(sp_time := DINT_TO_TIME(EDTP2S1_PARA_T1 * 1000),
						level_value := EDTLIT0604.status.value,
						set_point := EDTP2S1_PARA_L1,
						sp_accumulation := EDTP2S1_PARA_AC1,
						flowmeter := EDTFQIT0501,
						done := p2_step1_2_3_done);
						EDTP06.input.auto_run_signal := LiquidReleaseAdvanced_0.run;
						IF (NOT EDTP06.input.run_feedback) AND p2_step1_2_3_done AND (NOT EDTP06.input.auto_run_signal) THEN
							p2_step1_2_3_done := FALSE;
							p2_step1_2 := 4;
						END_IF;
					4:
						IF EDTFQIT0501.flowrate <= flowrate_threshold THEN
							EDTFQV0501.input.auto_open_signal := FALSE;
						END_IF;
						IF EDTFQV0501.input.close_feedback_state THEN
							p2_step1_2 := 5;
						END_IF;
					5:
						EDTXV0508.input.auto_open_signal := FALSE;
						IF EDTXV0508.input.close_feedback_state THEN
							EDTP2S1_STEP[2].done := TRUE;
							p2_step1_2 := 0;
						END_IF;
				END_CASE;
			3:
				EDTR01.input.auto_run_signal := TRUE;
				IF EDTTIT0501.status.value <= EDTP2S1_PARA_Temp1 THEN
					EDTXV0503.input.auto_open_signal := TRUE;
					IF EDTXV0503.input.open_feedback_state THEN
						EDTP05.input.auto_run_signal := TRUE;
						IF EDTP05.input.run_feedback THEN
							EDTP2S1_STEP[3].done := TRUE;
						END_IF;
					END_IF;
				END_IF;
			4:
				//人工抽入甲醇钠,此时需控制温度
				IF EDTTIT0501.status.value >= EDTP2S1_PARA_Temp2 THEN
					EDTXV0503.input.auto_open_signal := FALSE;
				END_IF;
				IF EDTTIT0501.status.value <= EDTP2S1_PARA_Temp3 THEN
					EDTXV0503.input.auto_open_signal := TRUE;
				END_IF;
			5:
				CASE p2_step1_5 OF
					0:
						IF NOT EDTP2S1_STEP[5].done THEN
							p2_step1_5 := 1;
						END_IF;
					1:
						EDTXV0501.input.auto_open_signal := FALSE;
						EDTXV0503.input.auto_open_signal := FALSE;
						EDTP05.input.auto_run_signal := FALSE;
						EDTPV0501.input.auto_open_signal := TRUE;
						p2_step1_5 := 2;
					2:
						IF EDTPIT0501.status.value >= EDTP2S1_PARA_P1 THEN
							EDTPV0501.input.auto_open_signal := FALSE;
							p2_step1_5 := 3;
						END_IF;
					3:
						TON_11.IN := TRUE;
						TON_11.PT := DINT_TO_TIME(EDTP2S1_PARA_T2 * 60 * 1000);
						IF TON_11.Q THEN
							TON_11.IN := FALSE;
							p2_step1_5 := 4;
						END_IF;
					4:
						EDTR01.input.auto_run_signal := FALSE;
						EDTXV0504.input.auto_open_signal := FALSE;
						p2_step1_5 := 0;
						EDTP2S1_STEP[5].done := TRUE;
				END_CASE;
				TON_11();
			6:
				//确认V13可以进料
			7:
				IF NOT EDTP2S1_STEP[7].done THEN
					EDTXV0507.input.auto_open_signal := TRUE;
					IF EDTPIT0501.status.value <= EDTP2S1_PARA_P2 THEN
						EDTPV0501.input.auto_open_signal := TRUE;
					END_IF;
					IF EDTPIT0501.status.value >= EDTP2S1_PARA_P3 THEN
						EDTPV0501.input.auto_open_signal := FALSE;
					END_IF;
				ELSE
					EDTXV0507.input.auto_open_signal := FALSE;
					EDTPV0501.input.auto_open_signal := FALSE;
				END_IF;
			8:
			//清理
		END_CASE;
	END_IF;

	//人工确认步骤可用
	IF (EDTP2S1.status.run_state) AND (NOT EDTP2S1_STEP[EDTP2S1.status.run_step].done AND ((EDTP2S1.status.run_step = 1) OR (EDTP2S1.status.run_step = 4) OR (EDTP2S1.status.run_step = 6)
		OR (EDTP2S1.status.run_step = 7) OR (EDTP2S1.status.run_step = 8))) THEN
		EDTP2S1.status.confirm_enable := TRUE;
	ELSE
		EDTP2S1.status.confirm_enable := FALSE;
	END_IF;
END_ACTION

(* ---- EDTP2S2A_ACTION.st ---- *)
ACTION P2S2A_ACT:
	//设定时间
	FOR i := 0 TO EDTP2S2_STEP_NUM DO
		IF EDTP2S2A_ST[i] < T#5s THEN
			EDTP2S2A_ST[i] := T#5s;
		END_IF;
		EDTP2S2A_STEP[i].set_time := EDTP2S2A_ST[i];
	END_FOR;

	//流程步骤
	ProcessHandleFC(EDTP2S2A,EDTP2S2A_STEP[0],EDTP2S2_STEP_NUM);

	//object 手自动切换
	IF (EDTP2S2A.status.mode <> 0) AND (NOT EDTP2S2A.auto_mode_edge) THEN
		EDTP2S2A.auto_mode_edge := TRUE;
		EDTP2S2A.manual_mode_edge := FALSE;

		EDTXV0601.control.auto_operate := TRUE;
		EDTP06.control.auto_operate := TRUE;
		EDTXV0603.control.auto_operate := TRUE;
		EDTP02.control.auto_operate := TRUE;
		EDTXV0602.control.auto_operate := TRUE;
		EDTP04.control.auto_operate := TRUE;
		EDTXV0609.control.auto_operate := TRUE;
		EDTXV0605.control.auto_operate := TRUE;
		EDTXV0606.control.auto_operate := TRUE;
		EDTXV0611.control.auto_operate := TRUE;
		EDTXV0645.control.auto_operate := TRUE;
		EDTR05A.control.auto_operate := TRUE;
		EDTXV0641.control.auto_operate := TRUE;
		EDTTV0601D.control.auto_operate := TRUE;
		EDTTV0601F.control.auto_operate := TRUE;
		EDTTV0601E.control.auto_operate := TRUE;
		EDTXV0604.control.auto_operate := TRUE;
		EDTXV0610.control.auto_operate := TRUE;
	END_IF;

	IF (EDTP2S2A.status.mode = 0) AND (NOT EDTP2S2A.manual_mode_edge) THEN
		EDTP2S2A.manual_mode_edge := TRUE;
		EDTP2S2A.auto_mode_edge := FALSE;

		EDTXV0601.control.manual_operate := TRUE;
		EDTP06.control.manual_operate := TRUE;
		EDTXV0603.control.manual_operate := TRUE;
		EDTP02.control.manual_operate := TRUE;
		EDTXV0602.control.manual_operate := TRUE;
		EDTP04.control.manual_operate := TRUE;
		EDTXV0609.control.manual_operate := TRUE;
		EDTXV0605.control.manual_operate := TRUE;
		EDTXV0606.control.manual_operate := TRUE;
		EDTXV0611.control.manual_operate := TRUE;
		EDTXV0645.control.manual_operate := TRUE;
		EDTR05A.control.manual_operate := TRUE;
		EDTXV0641.control.manual_operate := TRUE;
		EDTTV0601D.control.manual_operate := TRUE;
		EDTTV0601F.control.manual_operate := TRUE;
		EDTTV0601E.control.manual_operate := TRUE;
		EDTXV0604.control.manual_operate := TRUE;
		EDTXV0610.control.manual_operate := TRUE;
	END_IF;

	//错误信号停机
	EDTP2S2A.input.error_signal := (EDTXV0601.status.valve_status >= 2) OR (EDTP06.status.motor_status >= 2) OR
	(EDTXV0603.status.valve_status >= 2) OR(EDTP02.status.motor_status >= 2) OR (EDTXV0602.status.valve_status >= 2) OR
	(EDTP04.status.motor_status >= 2) OR (EDTXV0609.status.valve_status >= 2) OR (EDTXV0605.status.valve_status >= 2) OR
	(EDTXV0606.status.valve_status >= 2) OR (EDTXV0611.status.valve_status >= 2) OR (EDTXV0645.status.valve_status >= 2) OR
	(EDTR05A.status.motor_status >= 2) OR (EDTTV0601D.status.valve_status >= 2) OR (EDTXV0641.status.valve_status >= 2) OR
	(EDTTV0601F.status.valve_status >= 2) OR (EDTTV0601E.status.valve_status >= 2) OR (EDTXV0604.status.valve_status >= 2) OR (EDTXV0610.status.valve_status >= 2);

	IF EDTP2S2A.status.run_state = 1 THEN
		//步骤执行动作
		CASE EDTP2S2A.status.run_step OF
			0:
				//初始化
				IF NOT EDTP2S2A_STEP[0].done THEN
					EDTXV0601.control.auto_operate := TRUE;
					EDTP06.control.auto_operate := TRUE;
					EDTXV0603.control.auto_operate := TRUE;
					EDTP02.control.auto_operate := TRUE;
					EDTXV0602.control.auto_operate := TRUE;
					EDTP04.control.auto_operate := TRUE;
					EDTXV0609.control.auto_operate := TRUE;
					EDTXV0605.control.auto_operate := TRUE;
					EDTXV0606.control.auto_operate := TRUE;
					EDTXV0611.control.auto_operate := TRUE;
					EDTXV0645.control.auto_operate := TRUE;
					EDTR05A.control.auto_operate := TRUE;
					EDTXV0641.control.auto_operate := TRUE;
					EDTTV0601D.control.auto_operate := TRUE;
					EDTTV0601F.control.auto_operate := TRUE;
					EDTTV0601E.control.auto_operate := TRUE;
					EDTXV0604.control.auto_operate := TRUE;
					EDTXV0610.control.auto_operate := TRUE;
					EDTP2S2A_STEP[0].done := TRUE;
				END_IF;
			1:
				//人工投料edc
			2:
				EDTXV0610.input.auto_open_signal := FALSE;
				IF EDTXV0610.input.close_feedback_state THEN
					EDTXV0609.input.auto_open_signal := TRUE;
				END_IF;
				IF EDTXV0609.input.open_feedback_state THEN
					EDTXV0611.input.auto_open_signal := TRUE;
				END_IF;
				IF EDTXV0611.input.open_feedback_state THEN
					EDTXV0645.input.auto_open_signal := TRUE;
				END_IF;
				IF EDTXV0609.input.open_feedback_state AND EDTXV0611.input.open_feedback_state AND EDTXV0645.input.open_feedback_state THEN
					EDTP2S2A_STEP[2].done := TRUE;
				END_IF;
			3:
				CASE p2_step2_3a OF
					0:
						IF NOT EDTP2S2A_STEP[3].done THEN
							p2_step2_3a := 1;
						END_IF;
					1:
						EDTXV0605.input.auto_open_signal := TRUE;
						IF EDTXV0605.input.open_feedback_state THEN
							p2_step2_3a := 2;
						END_IF;
					2:
						TON_17.PT := DINT_TO_TIME(EDTP2S2_PARA_T4 * 60 * 1000);
						TON_17.IN := TRUE;
						IF TON_17.Q THEN
							TON_17.IN := FALSE;
							p2_step2_3a := 3;
						END_IF;
					3:
						EDTXV0606.input.auto_open_signal := TRUE;
						IF EDTXV0606.input.open_feedback_state THEN
							p2_step2_3a := 4;
						END_IF;
					4:
						TON_17.PT := DINT_TO_TIME(EDTP2S2_PARA_T5 * 60 * 1000);
						TON_17.IN := TRUE;
						IF TON_17.Q THEN
							TON_17.IN := FALSE;
							p2_step2_3a := 5;
						END_IF;
					5:
						EDTXV0605.input.auto_open_signal := FALSE;
						EDTXV0606.input.auto_open_signal := FALSE;
						IF EDTXV0605.input.close_feedback_state AND EDTXV0606.input.close_feedback_state THEN
							p2_step2_3a := 6;
						END_IF;
					6:
						p2_step2_3a := 7;
					7:
						IF EDTTIT0601.status.value < EDTP2S2_PARA_Temp1 THEN
							p2_step2_3a := 8;
						ELSE
							p2_step2_3a := 9;
						END_IF;
					8:
						//升温
						CASE p2_step2_3a_8 OF
							0:
								EDTTV0601F.input.auto_open_signal := TRUE;
								IF EDTTV0601F.input.open_feedback_state THEN
									EDTXV0641.input.auto_open_signal := TRUE;
									p2_step2_3a_8 := 1;
								END_IF;
							1:
								TON_8.PT := DINT_TO_TIME(EDTP2S2_PARA_T7 * 1000);
								TON_8.IN := TRUE;
								IF TON_8.Q THEN
									TON_8.IN := FALSE;
									p2_step2_3a_8 := 2;
								END_IF;
							2:
								EDTXV0641.input.auto_open_signal := FALSE;
								EDTTV0601F.input.auto_open_signal := FALSE;
								IF EDTTV0601F.input.close_feedback_state THEN
									p2_step2_3a_8 := 3;
								END_IF;
							3:
								EDTTV0601E.input.auto_open_signal := TRUE;
								IF EDTTV0601E.input.open_feedback_state THEN
									EDTTV0601D.input.auto_open_signal := TRUE;
									IF EDTTV0601D.input.open_feedback_state THEN
										p2_step2_3a_8 := 4;
									END_IF;
								END_IF;
							4:
								IF EDTTIT0601.status.value >= EDTP2S2_PARA_Temp1 THEN
									p2_step2_3a_8 := 5;
								END_IF;
							5:
								EDTTV0601D.input.auto_open_signal := FALSE;
								IF EDTTV0601D.input.close_feedback_state THEN
									EDTTV0601E.input.auto_open_signal := FALSE;
									IF EDTTV0601E.input.close_feedback_state THEN
										EDTTV0601F.input.auto_open_signal := TRUE;//21.2.5
										IF EDTTV0601F.input.open_feedback_state THEN
											p2_step2_3a_8 := 0;
											p2_step2_3a := 9;
										END_IF;
									END_IF;
								END_IF;
						END_CASE;
						TON_8();
					9:
						//温度和时间到enable confirm
						EDTR05A.input.auto_run_signal := TRUE;
						TON_17.PT := DINT_TO_TIME(EDTP2S2_PARA_T6 * 60 * 1000);
						TON_17.IN := TRUE;
						p2_step2_3a := 10;
					10:
						IF TON_17.Q THEN
							TON_17.IN := FALSE;
							p2_step2_3a_confirm_enable := TRUE;
						END_IF;
						IF EDTP2S2A_STEP[3].done THEN
							p2_step2_3a := 0;
							p2_step2_3a_confirm_enable := FALSE;
						END_IF;
				END_CASE;
				TON_17();
			4:
				CASE p2_step2_4a OF
					0:
						IF NOT EDTP2S2A_STEP[4].done THEN
							p2_step2_4a := 1;
						END_IF;
					1:
						EDTXV0604.input.auto_open_signal := TRUE;
						p2_step2_4a := 2;
					2:
						TON_15.PT := DINT_TO_TIME(EDTP2S2_PARA_T8 * 60 * 1000);
						TON_15.IN := TRUE;
						IF TON_15.Q THEN
							TON_15.IN := FALSE;
							p2_step2_4a := 3;
						END_IF;
					3:
						EDTXV0604.input.auto_open_signal := FALSE;
						IF EDTXV0604.input.close_feedback_state THEN
							p2_step2_4a := 4;
						END_IF;
					4:
						EDTTV0601F.input.auto_open_signal := TRUE;
						IF EDTTV0601F.input.open_feedback_state THEN
							EDTXV0641.input.auto_open_signal := TRUE;
							p2_step2_4a := 5;
						END_IF;
					5:
						TON_15.PT := DINT_TO_TIME(EDTP2S2_PARA_T7 * 1000);
						TON_15.IN := TRUE;
						IF TON_15.Q THEN
							TON_15.IN := FALSE;
							p2_step2_4a := 6;
						END_IF;
					6:
						EDTXV0641.input.auto_open_signal := FALSE;
						EDTTV0601F.input.auto_open_signal := FALSE;
						IF EDTTV0601F.input.close_feedback_state THEN
							p2_step2_4a := 7;
						END_IF;
					7:
						EDTTV0601E.input.auto_open_signal := TRUE;
						IF EDTTV0601E.input.open_feedback_state THEN
							EDTTV0601D.input.auto_open_signal := TRUE;
							IF EDTTV0601D.input.open_feedback_state THEN
								p2_step2_4a := 8;
							END_IF;
						END_IF;
					8:
						IF EDTTIT0601.status.value >= EDTP2S2_PARA_Temp2 THEN
							p2_step2_4a := 0;
							EDTP2S2A_STEP[4].done := TRUE;
						END_IF;
				END_CASE;
				TON_15();
			5:
				//确认回收结束
			6:
				EDTXV0609.input.auto_open_signal := FALSE;
				EDTXV0610.input.auto_open_signal := TRUE;
				EDTTV0601D.input.auto_open_signal := FALSE;
				IF EDTTV0601D.input.close_feedback_state THEN
					EDTTV0601E.input.auto_open_signal := FALSE;
					IF EDTTV0601E.input.close_feedback_state THEN
						EDTTV0601F.input.auto_open_signal := TRUE;//21.2.5
						IF EDTTV0601F.input.open_feedback_state THEN
							EDTP2S2A_STEP[6].done := TRUE;
						END_IF;
					END_IF;
				END_IF;
		END_CASE;
	END_IF;

	//V14进料
	IF v14_add THEN
		CASE v14_add_step OF
			0:
				EDTXV0601.input.auto_open_signal := TRUE;
				IF EDTXV0601.input.open_feedback_state THEN
					v14_add_step := 1;
				END_IF;
			1:
				LiquidTransfer_6(sp_time := DINT_TO_TIME(EDTP2S2_PARA_T1 * 1000),
				sp_accumulation := EDTP2S2_PARA_AC1,
				done := v14_add_step1_done,
				flowmeter := EDTFQIT0501);
				EDTP06.input.auto_run_signal := LiquidTransfer_6.run;
				IF v14_add_step1_done AND (NOT EDTP06.input.run_feedback) AND (NOT EDTP06.input.auto_run_signal)THEN
					v14_add_step := 2;
					v14_add_step1_done := FALSE;
				END_IF;
			2:
				IF EDTFQIT0501.flowrate <= flowrate_threshold THEN
					EDTXV0601.input.auto_open_signal := FALSE;
					v14_add_step := 0;
					v14_add := FALSE;
				END_IF;
		END_CASE;
	END_IF;
	//V15进料
	IF v15_add THEN
		CASE v15_add_step OF
			0:
				EDTXV0602.input.auto_open_signal := TRUE;
				IF EDTXV0602.input.open_feedback_state THEN
					v15_add_step := 1;
				END_IF;
			1:
				LiquidAddSimple_2(level_value := EDTLIT0602.status.value,
				sp_value := EDTP2S2_PARA_L1,
				sp_time := DINT_TO_TIME(EDTP2S2_PARA_T2 * 60 * 1000),
				done := v15_add_1_done);
				EDTP04.input.auto_run_signal := LiquidAddSimple_2.run;
				IF v15_add_1_done AND (NOT EDTP04.input.run_feedback) AND (NOT EDTP04.input.auto_run_signal) THEN
					v15_add_step := 2;
					v15_add_1_done := FALSE;
				END_IF;
			2:
				TON_12.PT := T#10s;
				TON_12.IN := TRUE;
				IF TON_12.Q THEN
					TON_12.IN := FALSE;
					v15_add_step := 3;
				END_IF;
			3:
				EDTXV0602.input.auto_open_signal := FALSE;
				v15_add_step := 0;
				v15_add := FALSE;
		END_CASE;
		TON_12();
	END_IF;
	//V16进料
	IF v16_add THEN
		CASE v16_add_step OF
			0:
				EDTXV0603.input.auto_open_signal := TRUE;
				IF EDTXV0603.input.open_feedback_state THEN
					v16_add_step := 1;
				END_IF;
			1:
				LiquidAddSimple_3(level_value := EDTLIT0603.status.value,
				sp_value := EDTP2S2_PARA_L2,
				sp_time := DINT_TO_TIME(EDTP2S2_PARA_T3 * 60 * 1000),
				done := v16_add_1_done);
				EDTP02.input.auto_run_signal := LiquidAddSimple_3.run;
				IF v16_add_1_done AND (NOT EDTP02.input.run_feedback) AND (NOT EDTP02.input.auto_run_signal) THEN
					v16_add_step := 2;
					v16_add_1_done := FALSE;
				END_IF;
			2:
				TON_14.PT := T#10s;
				TON_14.IN := TRUE;
				IF TON_14.Q THEN
					TON_14.IN := FALSE;
					v16_add_step := 3;
				END_IF;
			3:
				EDTXV0603.input.auto_open_signal := FALSE;
				v16_add_step := 0;
				v16_add := FALSE;
		END_CASE;
		TON_14();
	END_IF;

	//人工确认步骤可用
	IF (EDTP2S2A.status.run_state) AND (NOT EDTP2S2A_STEP[EDTP2S2A.status.run_step].done AND ((EDTP2S2A.status.run_step = 1) OR (EDTP2S2A.status.run_step = 5) OR (p2_step2_3a_confirm_enable))) THEN
		EDTP2S2A.status.confirm_enable := TRUE;
	ELSE
		EDTP2S2A.status.confirm_enable := FALSE;
	END_IF;
END_ACTION

(* ---- EDTP2S2B_ACTION.st ---- *)
ACTION P2S2B_ACT:
	//设定时间
	FOR i := 0 TO EDTP2S2_STEP_NUM DO
		IF EDTP2S2B_ST[i] < T#5s THEN
			EDTP2S2B_ST[i] := T#5s;
		END_IF;
		EDTP2S2B_STEP[i].set_time := EDTP2S2B_ST[i];
	END_FOR;

	//流程步骤
	ProcessHandleFC(EDTP2S2B,EDTP2S2B_STEP[0],EDTP2S2_STEP_NUM);

	//object 手自动切换
	IF (EDTP2S2B.status.mode <> 0) AND (NOT EDTP2S2B.auto_mode_edge) THEN
		EDTP2S2B.auto_mode_edge := TRUE;
		EDTP2S2B.manual_mode_edge := FALSE;

		EDTXV0601.control.auto_operate := TRUE;
		EDTP06.control.auto_operate := TRUE;
		EDTXV0603.control.auto_operate := TRUE;
		EDTP02.control.auto_operate := TRUE;
		EDTXV0602.control.auto_operate := TRUE;
		EDTP04.control.auto_operate := TRUE;
		EDTXV0621.control.auto_operate := TRUE;
		EDTXV0618.control.auto_operate := TRUE;
		EDTXV0619.control.auto_operate := TRUE;
		EDTXV0623.control.auto_operate := TRUE;
		EDTXV0645.control.auto_operate := TRUE;
		EDTR05B.control.auto_operate := TRUE;
		EDTXV0642.control.auto_operate := TRUE;
		EDTTV0603D.control.auto_operate := TRUE;
		EDTTV0603F.control.auto_operate := TRUE;
		EDTTV0603E.control.auto_operate := TRUE;
		EDTXV0617.control.auto_operate := TRUE;
		EDTXV0622.control.auto_operate := TRUE;
	END_IF;

	IF (EDTP2S2B.status.mode = 0) AND (NOT EDTP2S2B.manual_mode_edge) THEN
		EDTP2S2B.manual_mode_edge := TRUE;
		EDTP2S2B.auto_mode_edge := FALSE;

		EDTXV0601.control.manual_operate := TRUE;
		EDTP06.control.manual_operate := TRUE;
		EDTXV0603.control.manual_operate := TRUE;
		EDTP02.control.manual_operate := TRUE;
		EDTXV0602.control.manual_operate := TRUE;
		EDTP04.control.manual_operate := TRUE;
		EDTXV0621.control.manual_operate := TRUE;
		EDTXV0618.control.manual_operate := TRUE;
		EDTXV0619.control.manual_operate := TRUE;
		EDTXV0623.control.manual_operate := TRUE;
		EDTXV0645.control.manual_operate := TRUE;
		EDTR05B.control.manual_operate := TRUE;
		EDTXV0642.control.manual_operate := TRUE;
		EDTTV0603D.control.manual_operate := TRUE;
		EDTTV0603F.control.manual_operate := TRUE;
		EDTTV0603E.control.manual_operate := TRUE;
		EDTXV0617.control.manual_operate := TRUE;
		EDTXV0622.control.manual_operate := TRUE;
	END_IF;

	//错误信号停机
	EDTP2S2B.input.error_signal := (EDTXV0601.status.valve_status >= 2) OR (EDTP06.status.motor_status >= 2) OR
	(EDTXV0603.status.valve_status >= 2) OR(EDTP02.status.motor_status >= 2) OR (EDTXV0602.status.valve_status >= 2) OR
	(EDTP04.status.motor_status >= 2) OR (EDTXV0621.status.valve_status >= 2) OR (EDTXV0618.status.valve_status >= 2) OR
	(EDTXV0619.status.valve_status >= 2) OR (EDTXV0623.status.valve_status >= 2) OR (EDTXV0645.status.valve_status >= 2) OR
	(EDTR05B.status.motor_status >= 2) OR (EDTTV0603D.status.valve_status >= 2) OR (EDTXV0642.status.valve_status >= 2) OR
	(EDTTV0603F.status.valve_status >= 2) OR (EDTTV0603E.status.valve_status >= 2) OR (EDTXV0617.status.valve_status >= 2) OR (EDTXV0622.status.valve_status >= 2);

	IF EDTP2S2B.status.run_state = 1 THEN
		//步骤执行动作
		CASE EDTP2S2B.status.run_step OF
			0:
				//初始化
				IF NOT EDTP2S2B_STEP[0].done THEN
					EDTXV0601.control.auto_operate := TRUE;
					EDTP06.control.auto_operate := TRUE;
					EDTXV0603.control.auto_operate := TRUE;
					EDTP02.control.auto_operate := TRUE;
					EDTXV0602.control.auto_operate := TRUE;
					EDTP04.control.auto_operate := TRUE;
					EDTXV0621.control.auto_operate := TRUE;
					EDTXV0618.control.auto_operate := TRUE;
					EDTXV0619.control.auto_operate := TRUE;
					EDTXV0623.control.auto_operate := TRUE;
					EDTXV0645.control.auto_operate := TRUE;
					EDTR05B.control.auto_operate := TRUE;
					EDTXV0642.control.auto_operate := TRUE;
					EDTTV0603D.control.auto_operate := TRUE;
					EDTTV0603F.control.auto_operate := TRUE;
					EDTTV0603E.control.auto_operate := TRUE;
					EDTXV0617.control.auto_operate := TRUE;
					EDTXV0622.control.auto_operate := TRUE;
					EDTP2S2B_STEP[0].done := TRUE;
				END_IF;
			1:
				//人工投料edc
			2:
				EDTXV0622.input.auto_open_signal := FALSE;
				IF EDTXV0622.input.close_feedback_state THEN
					EDTXV0621.input.auto_open_signal := TRUE;
				END_IF;
				IF EDTXV0621.input.open_feedback_state THEN
					EDTXV0623.input.auto_open_signal := TRUE;
				END_IF;
				IF EDTXV0623.input.open_feedback_state THEN
					EDTXV0645.input.auto_open_signal := TRUE;
				END_IF;
				IF EDTXV0621.input.open_feedback_state AND EDTXV0623.input.open_feedback_state AND EDTXV0645.input.open_feedback_state THEN
					EDTP2S2B_STEP[2].done := TRUE;
				END_IF;
			3:
				CASE p2_step2_3b OF
					0:
						IF NOT EDTP2S2B_STEP[3].done THEN
							p2_step2_3b := 1;
						END_IF;
					1:
						EDTXV0618.input.auto_open_signal := TRUE;
						IF EDTXV0618.input.open_feedback_state THEN
							p2_step2_3b := 2;
						END_IF;
					2:
						TON_28.PT := DINT_TO_TIME(EDTP2S2_PARA_T4 * 60 * 1000);
						TON_28.IN := TRUE;
						IF TON_28.Q THEN
							TON_28.IN := FALSE;
							p2_step2_3b := 3;
						END_IF;
					3:
						EDTXV0619.input.auto_open_signal := TRUE;
						IF EDTXV0619.input.open_feedback_state THEN
							p2_step2_3b := 4;
						END_IF;
					4:
						TON_28.PT := DINT_TO_TIME(EDTP2S2_PARA_T5 * 60 * 1000);
						TON_28.IN := TRUE;
						IF TON_28.Q THEN
							TON_28.IN := FALSE;
							p2_step2_3b := 5;
						END_IF;
					5:
						EDTXV0618.input.auto_open_signal := FALSE;
						EDTXV0619.input.auto_open_signal := FALSE;
						IF EDTXV0618.input.close_feedback_state AND EDTXV0619.input.close_feedback_state THEN
							p2_step2_3b := 6;
						END_IF;
					6:
						p2_step2_3b := 7;
					7:
						IF EDTTIT0603.status.value < EDTP2S2_PARA_Temp1 THEN
							p2_step2_3b := 8;
						ELSE
							p2_step2_3b := 9;
						END_IF;
					8:
						//升温
						CASE p2_step2_3b_8 OF
							0:
								EDTTV0603F.input.auto_open_signal := TRUE;
								IF EDTTV0603F.input.open_feedback_state THEN
									EDTXV0642.input.auto_open_signal := TRUE;
									p2_step2_3b_8 := 1;
								END_IF;
							1:
								TON_30.PT := DINT_TO_TIME(EDTP2S2_PARA_T7 * 1000);
								TON_30.IN := TRUE;
								IF TON_30.Q THEN
									TON_30.IN := FALSE;
									p2_step2_3b_8 := 2;
								END_IF;
							2:
								EDTXV0642.input.auto_open_signal := FALSE;
								EDTTV0603F.input.auto_open_signal := FALSE;
								IF EDTTV0603F.input.close_feedback_state THEN
									p2_step2_3b_8 := 3;
								END_IF;
							3:
								EDTTV0603E.input.auto_open_signal := TRUE;
								IF EDTTV0603E.input.open_feedback_state THEN
									EDTTV0603D.input.auto_open_signal := TRUE;
									IF EDTTV0603D.input.open_feedback_state THEN
										p2_step2_3b_8 := 4;
									END_IF;
								END_IF;
							4:
								IF EDTTIT0603.status.value >= EDTP2S2_PARA_Temp1 THEN
									p2_step2_3b_8 := 5;
								END_IF;
							5:
								EDTTV0603D.input.auto_open_signal := FALSE;
								IF EDTTV0603D.input.close_feedback_state THEN
									EDTTV0603E.input.auto_open_signal := FALSE;
									IF EDTTV0603E.input.close_feedback_state THEN
										EDTTV0603F.input.auto_open_signal := TRUE;//21.2.5
										IF EDTTV0603F.input.open_feedback_state THEN
											p2_step2_3b_8 := 0;
											p2_step2_3b := 9;
										END_IF;
									END_IF;
								END_IF;
						END_CASE;
						TON_30();
					9:
						//温度和时间到enable confirm
						EDTR05B.input.auto_run_signal := TRUE;
						TON_28.PT := DINT_TO_TIME(EDTP2S2_PARA_T6 * 60 * 1000);
						TON_28.IN := TRUE;
						p2_step2_3b := 10;
					10:
						IF TON_28.Q THEN
							TON_28.IN := FALSE;
							p2_step2_3b_confirm_enable := TRUE;
						END_IF;
						IF EDTP2S2B_STEP[3].done THEN
							p2_step2_3b := 0;
							p2_step2_3b_confirm_enable := FALSE;
						END_IF;
				END_CASE;
				TON_28();
			4:
				CASE p2_step2_4b OF
					0:
						IF NOT EDTP2S2B_STEP[4].done THEN
							p2_step2_4b := 1;
						END_IF;
					1:
						EDTXV0617.input.auto_open_signal := TRUE;
						p2_step2_4b := 2;
					2:
						TON_31.PT := DINT_TO_TIME(EDTP2S2_PARA_T8 * 60 * 1000);
						TON_31.IN := TRUE;
						IF TON_31.Q THEN
							TON_31.IN := FALSE;
							p2_step2_4b := 3;
						END_IF;
					3:
						EDTXV0617.input.auto_open_signal := FALSE;
						IF EDTXV0617.input.close_feedback_state THEN
							p2_step2_4b := 4;
						END_IF;
					4:
						EDTTV0603F.input.auto_open_signal := TRUE;
						IF EDTTV0603F.input.open_feedback_state THEN
							EDTXV0642.input.auto_open_signal := TRUE;
							p2_step2_4b := 5;
						END_IF;
					5:
						TON_31.PT := DINT_TO_TIME(EDTP2S2_PARA_T7 * 1000);
						TON_31.IN := TRUE;
						IF TON_31.Q THEN
							TON_31.IN := FALSE;
							p2_step2_4b := 6;
						END_IF;
					6:
						EDTXV0642.input.auto_open_signal := FALSE;
						EDTTV0603F.input.auto_open_signal := FALSE;
						IF EDTTV0603F.input.close_feedback_state THEN
							p2_step2_4b := 7;
						END_IF;
					7:
						EDTTV0603E.input.auto_open_signal := TRUE;
						IF EDTTV0603E.input.open_feedback_state THEN
							EDTTV0603D.input.auto_open_signal := TRUE;
							IF EDTTV0603D.input.open_feedback_state THEN
								p2_step2_4b := 8;
							END_IF;
						END_IF;
					8:
						IF EDTTIT0603.status.value >= EDTP2S2_PARA_Temp2 THEN
							p2_step2_4b := 0;
							EDTP2S2B_STEP[4].done := TRUE;
						END_IF;
				END_CASE;
				TON_31();
			5:
				//确认回收结束
			6:
				EDTXV0621.input.auto_open_signal := FALSE;
				EDTXV0622.input.auto_open_signal := TRUE;
				EDTTV0603D.input.auto_open_signal := FALSE;
				IF EDTTV0603D.input.close_feedback_state THEN
					EDTTV0603E.input.auto_open_signal := FALSE;
					IF EDTTV0603E.input.close_feedback_state THEN
						EDTTV0603F.input.auto_open_signal := TRUE;//21.2.5
						IF EDTTV0603F.input.open_feedback_state THEN
							EDTP2S2B_STEP[6].done := TRUE;
						END_IF;
					END_IF;
				END_IF;
		END_CASE;
	END_IF;

	//人工确认步骤可用
	IF (EDTP2S2B.status.run_state) AND (NOT EDTP2S2B_STEP[EDTP2S2B.status.run_step].done AND ((EDTP2S2B.status.run_step = 1) OR (EDTP2S2B.status.run_step = 5) OR (p2_step2_3b_confirm_enable))) THEN
		EDTP2S2B.status.confirm_enable := TRUE;
	ELSE
		EDTP2S2B.status.confirm_enable := FALSE;
	END_IF;
END_ACTION

(* ---- EDTP2S2C_ACTION.st ---- *)
ACTION P2S2C_ACT:
	//设定时间
	FOR i := 0 TO EDTP2S2_STEP_NUM DO
		IF EDTP2S2C_ST[i] < T#5s THEN
			EDTP2S2C_ST[i] := T#5s;
		END_IF;
		EDTP2S2C_STEP[i].set_time := EDTP2S2C_ST[i];
	END_FOR;

	//流程步骤
	ProcessHandleFC(EDTP2S2C,EDTP2S2C_STEP[0],EDTP2S2_STEP_NUM);

	//object 手自动切换
	IF (EDTP2S2C.status.mode <> 0) AND (NOT EDTP2S2C.auto_mode_edge) THEN
		EDTP2S2C.auto_mode_edge := TRUE;
		EDTP2S2C.manual_mode_edge := FALSE;

		EDTXV0601.control.auto_operate := TRUE;
		EDTP06.control.auto_operate := TRUE;
		EDTXV0603.control.auto_operate := TRUE;
		EDTP02.control.auto_operate := TRUE;
		EDTXV0602.control.auto_operate := TRUE;
		EDTP04.control.auto_operate := TRUE;
		EDTXV0629.control.auto_operate := TRUE;
		EDTXV0626.control.auto_operate := TRUE;
		EDTXV0627.control.auto_operate := TRUE;
		EDTXV0631.control.auto_operate := TRUE;
		EDTXV0645.control.auto_operate := TRUE;
		EDTR05C.control.auto_operate := TRUE;
		EDTXV0643.control.auto_operate := TRUE;
		EDTTV0605D.control.auto_operate := TRUE;
		EDTTV0605F.control.auto_operate := TRUE;
		EDTTV0605E.control.auto_operate := TRUE;
		EDTXV0625.control.auto_operate := TRUE;
		EDTXV0630.control.auto_operate := TRUE;
	END_IF;

	IF (EDTP2S2C.status.mode = 0) AND (NOT EDTP2S2C.manual_mode_edge) THEN
		EDTP2S2C.manual_mode_edge := TRUE;
		EDTP2S2C.auto_mode_edge := FALSE;

		EDTXV0601.control.manual_operate := TRUE;
		EDTP06.control.manual_operate := TRUE;
		EDTXV0603.control.manual_operate := TRUE;
		EDTP02.control.manual_operate := TRUE;
		EDTXV0602.control.manual_operate := TRUE;
		EDTP04.control.manual_operate := TRUE;
		EDTXV0629.control.manual_operate := TRUE;
		EDTXV0626.control.manual_operate := TRUE;
		EDTXV0627.control.manual_operate := TRUE;
		EDTXV0631.control.manual_operate := TRUE;
		EDTXV0645.control.manual_operate := TRUE;
		EDTR05C.control.manual_operate := TRUE;
		EDTXV0643.control.manual_operate := TRUE;
		EDTTV0605D.control.manual_operate := TRUE;
		EDTTV0605F.control.manual_operate := TRUE;
		EDTTV0605E.control.manual_operate := TRUE;
		EDTXV0625.control.manual_operate := TRUE;
		EDTXV0630.control.manual_operate := TRUE;
	END_IF;

	//错误信号停机
	EDTP2S2C.input.error_signal := (EDTXV0601.status.valve_status >= 2) OR (EDTP06.status.motor_status >= 2) OR
	(EDTXV0603.status.valve_status >= 2) OR(EDTP02.status.motor_status >= 2) OR (EDTXV0602.status.valve_status >= 2) OR
	(EDTP04.status.motor_status >= 2) OR (EDTXV0629.status.valve_status >= 2) OR (EDTXV0626.status.valve_status >= 2) OR
	(EDTXV0627.status.valve_status >= 2) OR (EDTXV0631.status.valve_status >= 2) OR (EDTXV0645.status.valve_status >= 2) OR
	(EDTR05C.status.motor_status >= 2) OR (EDTTV0605D.status.valve_status >= 2) OR (EDTXV0643.status.valve_status >= 2) OR
	(EDTTV0605F.status.valve_status >= 2) OR (EDTTV0605E.status.valve_status >= 2) OR (EDTXV0625.status.valve_status >= 2) OR (EDTXV0630.status.valve_status >= 2);

	IF EDTP2S2C.status.run_state = 1 THEN
		//步骤执行动作
		CASE EDTP2S2C.status.run_step OF
			0:
				//初始化
				IF NOT EDTP2S2C_STEP[0].done THEN
					EDTXV0601.control.auto_operate := TRUE;
					EDTP06.control.auto_operate := TRUE;
					EDTXV0603.control.auto_operate := TRUE;
					EDTP02.control.auto_operate := TRUE;
					EDTXV0602.control.auto_operate := TRUE;
					EDTP04.control.auto_operate := TRUE;
					EDTXV0629.control.auto_operate := TRUE;
					EDTXV0626.control.auto_operate := TRUE;
					EDTXV0627.control.auto_operate := TRUE;
					EDTXV0631.control.auto_operate := TRUE;
					EDTXV0645.control.auto_operate := TRUE;
					EDTR05C.control.auto_operate := TRUE;
					EDTXV0643.control.auto_operate := TRUE;
					EDTTV0605D.control.auto_operate := TRUE;
					EDTTV0605F.control.auto_operate := TRUE;
					EDTTV0605E.control.auto_operate := TRUE;
					EDTXV0625.control.auto_operate := TRUE;
					EDTXV0630.control.auto_operate := TRUE;
					EDTP2S2C_STEP[0].done := TRUE;
				END_IF;
			1:
				//人工投料edc
			2:
				EDTXV0630.input.auto_open_signal := FALSE;
				IF EDTXV0630.input.close_feedback_state THEN
					EDTXV0629.input.auto_open_signal := TRUE;
				END_IF;
				IF EDTXV0629.input.open_feedback_state THEN
					EDTXV0631.input.auto_open_signal := TRUE;
				END_IF;
				IF EDTXV0631.input.open_feedback_state THEN
					EDTXV0645.input.auto_open_signal := TRUE;
				END_IF;
				IF EDTXV0629.input.open_feedback_state AND EDTXV0631.input.open_feedback_state AND EDTXV0645.input.open_feedback_state THEN
					EDTP2S2C_STEP[2].done := TRUE;
				END_IF;
			3:
				CASE p2_step2_3c OF
					0:
						IF NOT EDTP2S2C_STEP[3].done THEN
							p2_step2_3c := 1;
						END_IF;
					1:
						EDTXV0626.input.auto_open_signal := TRUE;
						IF EDTXV0626.input.open_feedback_state THEN
							p2_step2_3c := 2;
						END_IF;
					2:
						TON_32.PT := DINT_TO_TIME(EDTP2S2_PARA_T4 * 60 * 1000);
						TON_32.IN := TRUE;
						IF TON_32.Q THEN
							TON_32.IN := FALSE;
							p2_step2_3c := 3;
						END_IF;
					3:
						EDTXV0627.input.auto_open_signal := TRUE;
						IF EDTXV0627.input.open_feedback_state THEN
							p2_step2_3c := 4;
						END_IF;
					4:
						TON_32.PT := DINT_TO_TIME(EDTP2S2_PARA_T5 * 60 * 1000);
						TON_32.IN := TRUE;
						IF TON_32.Q THEN
							TON_32.IN := FALSE;
							p2_step2_3c := 5;
						END_IF;
					5:
						EDTXV0626.input.auto_open_signal := FALSE;
						EDTXV0627.input.auto_open_signal := FALSE;
						IF EDTXV0626.input.close_feedback_state AND EDTXV0627.input.close_feedback_state THEN
							p2_step2_3c := 6;
						END_IF;
					6:
						p2_step2_3c := 7;
					7:
						IF EDTTIT0605.status.value < EDTP2S2_PARA_Temp1 THEN
							p2_step2_3c := 8;
						ELSE
							p2_step2_3c := 9;
						END_IF;
					8:
						//升温
						CASE p2_step2_3c_8 OF
							0:
								EDTTV0605F.input.auto_open_signal := TRUE;
								IF EDTTV0605F.input.open_feedback_state THEN
									EDTXV0643.input.auto_open_signal := TRUE;
									p2_step2_3c_8 := 1;
								END_IF;
							1:
								TON_33.PT := DINT_TO_TIME(EDTP2S2_PARA_T7 * 1000);
								TON_33.IN := TRUE;
								IF TON_33.Q THEN
									TON_33.IN := FALSE;
									p2_step2_3c_8 := 2;
								END_IF;
							2:
								EDTXV0643.input.auto_open_signal := FALSE;
								EDTTV0605F.input.auto_open_signal := FALSE;
								IF EDTTV0605F.input.close_feedback_state THEN
									p2_step2_3c_8 := 3;
								END_IF;
							3:
								EDTTV0605E.input.auto_open_signal := TRUE;
								IF EDTTV0605E.input.open_feedback_state THEN
									EDTTV0605D.input.auto_open_signal := TRUE;
									IF EDTTV0605D.input.open_feedback_state THEN
										p2_step2_3c_8 := 4;
									END_IF;
								END_IF;
							4:
								IF EDTTIT0605.status.value >= EDTP2S2_PARA_Temp1 THEN
									p2_step2_3c_8 := 5;
								END_IF;
							5:
								EDTTV0605D.input.auto_open_signal := FALSE;
								IF EDTTV0605D.input.close_feedback_state THEN
									EDTTV0605E.input.auto_open_signal := FALSE;
									IF EDTTV0605E.input.close_feedback_state THEN
										EDTTV0605F.input.auto_open_signal := TRUE;//21.2.5
										IF EDTTV0605F.input.open_feedback_state THEN
											p2_step2_3c_8 := 0;
											p2_step2_3c := 9;
										END_IF;
									END_IF;
								END_IF;
						END_CASE;
						TON_33();
					9:
						//温度和时间到enable confirm
						EDTR05C.input.auto_run_signal := TRUE;
						TON_32.PT := DINT_TO_TIME(EDTP2S2_PARA_T6 * 60 * 1000);
						TON_32.IN := TRUE;
						p2_step2_3c := 10;
					10:
						IF TON_32.Q THEN
							TON_32.IN := FALSE;
							p2_step2_3c_confirm_enable := TRUE;
						END_IF;
						IF EDTP2S2C_STEP[3].done THEN
							p2_step2_3c := 0;
							p2_step2_3c_confirm_enable := FALSE;
						END_IF;
				END_CASE;
				TON_32();
			4:
				CASE p2_step2_4c OF
					0:
						IF NOT EDTP2S2C_STEP[4].done THEN
							p2_step2_4c := 1;
						END_IF;
					1:
						EDTXV0625.input.auto_open_signal := TRUE;
						p2_step2_4c := 2;
					2:
						TON_34.PT := DINT_TO_TIME(EDTP2S2_PARA_T8 * 60 * 1000);
						TON_34.IN := TRUE;
						IF TON_34.Q THEN
							TON_34.IN := FALSE;
							p2_step2_4c := 3;
						END_IF;
					3:
						EDTXV0625.input.auto_open_signal := FALSE;
						IF EDTXV0625.input.close_feedback_state THEN
							p2_step2_4c := 4;
						END_IF;
					4:
						EDTTV0605F.input.auto_open_signal := TRUE;
						IF EDTTV0605F.input.open_feedback_state THEN
							EDTXV0643.input.auto_open_signal := TRUE;
							p2_step2_4c := 5;
						END_IF;
					5:
						TON_34.PT := DINT_TO_TIME(EDTP2S2_PARA_T7 * 1000);
						TON_34.IN := TRUE;
						IF TON_34.Q THEN
							TON_34.IN := FALSE;
							p2_step2_4c := 6;
						END_IF;
					6:
						EDTXV0643.input.auto_open_signal := FALSE;
						EDTTV0605F.input.auto_open_signal := FALSE;
						IF EDTTV0605F.input.close_feedback_state THEN
							p2_step2_4c := 7;
						END_IF;
					7:
						EDTTV0605E.input.auto_open_signal := TRUE;
						IF EDTTV0605E.input.open_feedback_state THEN
							EDTTV0605D.input.auto_open_signal := TRUE;
							IF EDTTV0605D.input.open_feedback_state THEN
								p2_step2_4c := 8;
							END_IF;
						END_IF;
					8:
						IF EDTTIT0605.status.value >= EDTP2S2_PARA_Temp2 THEN
							p2_step2_4c := 0;
							EDTP2S2C_STEP[4].done := TRUE;
						END_IF;
				END_CASE;
				TON_34();
			5:
				//确认回收结束
			6:
				EDTXV0629.input.auto_open_signal := FALSE;
				EDTXV0630.input.auto_open_signal := TRUE;
				EDTTV0605D.input.auto_open_signal := FALSE;
				IF EDTTV0605D.input.close_feedback_state THEN
					EDTTV0605E.input.auto_open_signal := FALSE;
					IF EDTTV0605E.input.close_feedback_state THEN
						EDTTV0605F.input.auto_open_signal := TRUE;//21.2.5
						IF EDTTV0605F.input.open_feedback_state THEN
							EDTP2S2C_STEP[6].done := TRUE;
						END_IF;
					END_IF;
				END_IF;
		END_CASE;
	END_IF;

	//人工确认步骤可用
	IF (EDTP2S2C.status.run_state) AND (NOT EDTP2S2C_STEP[EDTP2S2C.status.run_step].done AND ((EDTP2S2C.status.run_step = 1) OR (EDTP2S2C.status.run_step = 5) OR (p2_step2_3c_confirm_enable))) THEN
		EDTP2S2C.status.confirm_enable := TRUE;
	ELSE
		EDTP2S2C.status.confirm_enable := FALSE;
	END_IF;
END_ACTION

(* ---- EDTP2S2D_ACTION.st ---- *)
ACTION P2S2D_ACT:
	//设定时间
	FOR i := 0 TO EDTP2S2_STEP_NUM DO
		IF EDTP2S2D_ST[i] < T#5s THEN
			EDTP2S2D_ST[i] := T#5s;
		END_IF;
		EDTP2S2D_STEP[i].set_time := EDTP2S2D_ST[i];
	END_FOR;

	//流程步骤
	ProcessHandleFC(EDTP2S2D,EDTP2S2D_STEP[0],EDTP2S2_STEP_NUM);

	//object 手自动切换
	IF (EDTP2S2D.status.mode <> 0) AND (NOT EDTP2S2D.auto_mode_edge) THEN
		EDTP2S2D.auto_mode_edge := TRUE;
		EDTP2S2D.manual_mode_edge := FALSE;

		EDTXV0601.control.auto_operate := TRUE;
		EDTP06.control.auto_operate := TRUE;
		EDTXV0603.control.auto_operate := TRUE;
		EDTP02.control.auto_operate := TRUE;
		EDTXV0602.control.auto_operate := TRUE;
		EDTP04.control.auto_operate := TRUE;
		EDTXV0637.control.auto_operate := TRUE;
		EDTXV0634.control.auto_operate := TRUE;
		EDTXV0635.control.auto_operate := TRUE;
		EDTXV0639.control.auto_operate := TRUE;
		EDTXV0645.control.auto_operate := TRUE;
		EDTR05D.control.auto_operate := TRUE;
		EDTXV0644.control.auto_operate := TRUE;
		EDTTV0607D.control.auto_operate := TRUE;
		EDTTV0607F.control.auto_operate := TRUE;
		EDTTV0607E.control.auto_operate := TRUE;
		EDTXV0633.control.auto_operate := TRUE;
		EDTXV0638.control.auto_operate := TRUE;
	END_IF;

	IF (EDTP2S2D.status.mode = 0) AND (NOT EDTP2S2D.manual_mode_edge) THEN
		EDTP2S2D.manual_mode_edge := TRUE;
		EDTP2S2D.auto_mode_edge := FALSE;

		EDTXV0601.control.manual_operate := TRUE;
		EDTP06.control.manual_operate := TRUE;
		EDTXV0603.control.manual_operate := TRUE;
		EDTP02.control.manual_operate := TRUE;
		EDTXV0602.control.manual_operate := TRUE;
		EDTP04.control.manual_operate := TRUE;
		EDTXV0637.control.manual_operate := TRUE;
		EDTXV0634.control.manual_operate := TRUE;
		EDTXV0635.control.manual_operate := TRUE;
		EDTXV0639.control.manual_operate := TRUE;
		EDTXV0645.control.manual_operate := TRUE;
		EDTR05D.control.manual_operate := TRUE;
		EDTXV0644.control.manual_operate := TRUE;
		EDTTV0607D.control.manual_operate := TRUE;
		EDTTV0607F.control.manual_operate := TRUE;
		EDTTV0607E.control.manual_operate := TRUE;
		EDTXV0633.control.manual_operate := TRUE;
		EDTXV0638.control.manual_operate := TRUE;
	END_IF;

	//错误信号停机
	EDTP2S2D.input.error_signal := (EDTXV0601.status.valve_status >= 2) OR (EDTP06.status.motor_status >= 2) OR
	(EDTXV0603.status.valve_status >= 2) OR(EDTP02.status.motor_status >= 2) OR (EDTXV0602.status.valve_status >= 2) OR
	(EDTP04.status.motor_status >= 2) OR (EDTXV0637.status.valve_status >= 2) OR (EDTXV0634.status.valve_status >= 2) OR
	(EDTXV0635.status.valve_status >= 2) OR (EDTXV0639.status.valve_status >= 2) OR (EDTXV0645.status.valve_status >= 2) OR
	(EDTR05D.status.motor_status >= 2) OR (EDTTV0607D.status.valve_status >= 2) OR (EDTXV0644.status.valve_status >= 2) OR
	(EDTTV0607F.status.valve_status >= 2) OR (EDTTV0607E.status.valve_status >= 2) OR (EDTXV0633.status.valve_status >= 2) OR (EDTXV0638.status.valve_status >= 2);

	IF EDTP2S2D.status.run_state = 1 THEN
		//步骤执行动作
		CASE EDTP2S2D.status.run_step OF
			0:
				//初始化
				IF NOT EDTP2S2D_STEP[0].done THEN
					EDTXV0601.control.auto_operate := TRUE;
					EDTP06.control.auto_operate := TRUE;
					EDTXV0603.control.auto_operate := TRUE;
					EDTP02.control.auto_operate := TRUE;
					EDTXV0602.control.auto_operate := TRUE;
					EDTP04.control.auto_operate := TRUE;
					EDTXV0637.control.auto_operate := TRUE;
					EDTXV0634.control.auto_operate := TRUE;
					EDTXV0635.control.auto_operate := TRUE;
					EDTXV0639.control.auto_operate := TRUE;
					EDTXV0645.control.auto_operate := TRUE;
					EDTR05D.control.auto_operate := TRUE;
					EDTXV0644.control.auto_operate := TRUE;
					EDTTV0607D.control.auto_operate := TRUE;
					EDTTV0607F.control.auto_operate := TRUE;
					EDTTV0607E.control.auto_operate := TRUE;
					EDTXV0633.control.auto_operate := TRUE;
					EDTXV0638.control.auto_operate := TRUE;
					EDTP2S2D_STEP[0].done := TRUE;
				END_IF;
			1:
				//人工投料edc
			2:
				EDTXV0638.input.auto_open_signal := FALSE;
				IF EDTXV0638.input.close_feedback_state THEN
					EDTXV0637.input.auto_open_signal := TRUE;
				END_IF;
				IF EDTXV0637.input.open_feedback_state THEN
					EDTXV0639.input.auto_open_signal := TRUE;
				END_IF;
				IF EDTXV0639.input.open_feedback_state THEN
					EDTXV0645.input.auto_open_signal := TRUE;
				END_IF;
				IF EDTXV0637.input.open_feedback_state AND EDTXV0639.input.open_feedback_state AND EDTXV0645.input.open_feedback_state THEN
					EDTP2S2D_STEP[2].done := TRUE;
				END_IF;
			3:
				CASE p2_step2_3d OF
					0:
						IF NOT EDTP2S2D_STEP[3].done THEN
							p2_step2_3d := 1;
						END_IF;
					1:
						EDTXV0634.input.auto_open_signal := TRUE;
						IF EDTXV0634.input.open_feedback_state THEN
							p2_step2_3d := 2;
						END_IF;
					2:
						TON_35.PT := DINT_TO_TIME(EDTP2S2_PARA_T4 * 60 * 1000);
						TON_35.IN := TRUE;
						IF TON_35.Q THEN
							TON_35.IN := FALSE;
							p2_step2_3d := 3;
						END_IF;
					3:
						EDTXV0635.input.auto_open_signal := TRUE;
						IF EDTXV0635.input.open_feedback_state THEN
							p2_step2_3d := 4;
						END_IF;
					4:
						TON_35.PT := DINT_TO_TIME(EDTP2S2_PARA_T5 * 60 * 1000);
						TON_35.IN := TRUE;
						IF TON_35.Q THEN
							TON_35.IN := FALSE;
							p2_step2_3d := 5;
						END_IF;
					5:
						EDTXV0634.input.auto_open_signal := FALSE;
						EDTXV0635.input.auto_open_signal := FALSE;
						IF EDTXV0634.input.close_feedback_state AND EDTXV0635.input.close_feedback_state THEN
							p2_step2_3d := 6;
						END_IF;
					6:
						p2_step2_3d := 7;
					7:
						IF EDTTIT0607.status.value < EDTP2S2_PARA_Temp1 THEN
							p2_step2_3d := 8;
						ELSE
							p2_step2_3d := 9;
						END_IF;
					8:
						//升温
						CASE p2_step2_3d_8 OF
							0:
								EDTTV0607F.input.auto_open_signal := TRUE;
								IF EDTTV0607F.input.open_feedback_state THEN
									EDTXV0644.input.auto_open_signal := TRUE;
									p2_step2_3d_8 := 1;
								END_IF;
							1:
								TON_36.PT := DINT_TO_TIME(EDTP2S2_PARA_T7 * 1000);
								TON_36.IN := TRUE;
								IF TON_36.Q THEN
									TON_36.IN := FALSE;
									p2_step2_3d_8 := 2;
								END_IF;
							2:
								EDTXV0644.input.auto_open_signal := FALSE;
								EDTTV0607F.input.auto_open_signal := FALSE;
								IF EDTTV0607F.input.close_feedback_state THEN
									p2_step2_3d_8 := 3;
								END_IF;
							3:
								EDTTV0607E.input.auto_open_signal := TRUE;
								IF EDTTV0607E.input.open_feedback_state THEN
									EDTTV0607D.input.auto_open_signal := TRUE;
									IF EDTTV0607D.input.open_feedback_state THEN
										p2_step2_3d_8 := 4;
									END_IF;
								END_IF;
							4:
								IF EDTTIT0607.status.value >= EDTP2S2_PARA_Temp1 THEN
									p2_step2_3d_8 := 5;
								END_IF;
							5:
								EDTTV0607D.input.auto_open_signal := FALSE;
								IF EDTTV0607D.input.close_feedback_state THEN
									EDTTV0607E.input.auto_open_signal := FALSE;
									IF EDTTV0607E.input.close_feedback_state THEN
										EDTTV0607F.input.auto_open_signal := TRUE;//21.2.5
										IF EDTTV0607F.input.open_feedback_state THEN
											p2_step2_3d_8 := 0;
											p2_step2_3d := 9;
										END_IF;
									END_IF;
								END_IF;
						END_CASE;
						TON_36();
					9:
						//温度和时间到enable confirm
						EDTR05D.input.auto_run_signal := TRUE;
						TON_35.PT := DINT_TO_TIME(EDTP2S2_PARA_T6 * 60 * 1000);
						TON_35.IN := TRUE;
						p2_step2_3d := 10;
					10:
						IF TON_35.Q THEN
							TON_35.IN := FALSE;
							p2_step2_3d_confirm_enable := TRUE;
						END_IF;
						IF EDTP2S2D_STEP[3].done THEN
							p2_step2_3d := 0;
							p2_step2_3d_confirm_enable := FALSE;
						END_IF;
				END_CASE;
				TON_35();
			4:
				CASE p2_step2_4d OF
					0:
						IF NOT EDTP2S2D_STEP[4].done THEN
							p2_step2_4d := 1;
						END_IF;
					1:
						EDTXV0633.input.auto_open_signal := TRUE;
						p2_step2_4d := 2;
					2:
						TON_37.PT := DINT_TO_TIME(EDTP2S2_PARA_T8 * 60 * 1000);
						TON_37.IN := TRUE;
						IF TON_37.Q THEN
							TON_37.IN := FALSE;
							p2_step2_4d := 3;
						END_IF;
					3:
						EDTXV0633.input.auto_open_signal := FALSE;
						IF EDTXV0633.input.close_feedback_state THEN
							p2_step2_4d := 4;
						END_IF;
					4:
						EDTTV0607F.input.auto_open_signal := TRUE;
						IF EDTTV0607F.input.open_feedback_state THEN
							EDTXV0644.input.auto_open_signal := TRUE;
							p2_step2_4d := 5;
						END_IF;
					5:
						TON_37.PT := DINT_TO_TIME(EDTP2S2_PARA_T7 * 1000);
						TON_37.IN := TRUE;
						IF TON_37.Q THEN
							TON_37.IN := FALSE;
							p2_step2_4d := 6;
						END_IF;
					6:
						EDTXV0644.input.auto_open_signal := FALSE;
						EDTTV0607F.input.auto_open_signal := FALSE;
						IF EDTTV0607F.input.close_feedback_state THEN
							p2_step2_4d := 7;
						END_IF;
					7:
						EDTTV0607E.input.auto_open_signal := TRUE;
						IF EDTTV0607E.input.open_feedback_state THEN
							EDTTV0607D.input.auto_open_signal := TRUE;
							IF EDTTV0607D.input.open_feedback_state THEN
								p2_step2_4d := 8;
							END_IF;
						END_IF;
					8:
						IF EDTTIT0607.status.value >= EDTP2S2_PARA_Temp2 THEN
							p2_step2_4d := 0;
							EDTP2S2D_STEP[4].done := TRUE;
						END_IF;
				END_CASE;
				TON_37();
			5:
				//确认回收结束
			6:
				EDTXV0637.input.auto_open_signal := FALSE;
				EDTXV0638.input.auto_open_signal := TRUE;
				EDTTV0607D.input.auto_open_signal := FALSE;
				IF EDTTV0607D.input.close_feedback_state THEN
					EDTTV0607E.input.auto_open_signal := FALSE;
					IF EDTTV0607E.input.close_feedback_state THEN
						EDTTV0607F.input.auto_open_signal := TRUE;//21.2.5
						IF EDTTV0607F.input.open_feedback_state THEN
							EDTP2S2D_STEP[6].done := TRUE;
						END_IF;
					END_IF;
				END_IF;
		END_CASE;
	END_IF;

	//人工确认步骤可用
	IF (EDTP2S2D.status.run_state) AND (NOT EDTP2S2D_STEP[EDTP2S2D.status.run_step].done AND ((EDTP2S2D.status.run_step = 1) OR (EDTP2S2D.status.run_step = 5) OR (p2_step2_3d_confirm_enable))) THEN
		EDTP2S2D.status.confirm_enable := TRUE;
	ELSE
		EDTP2S2D.status.confirm_enable := FALSE;
	END_IF;
END_ACTION
